VAR_INPUT
  ENCODER : DINT ;	//Positionswert Encoder
  INKR : DINT ;	//Inkremente für einen gezählten Wegimpuls (TEILUNG)
  FRG : BOOL ;	//Zählfreigabe
  RICHTUNG : BOOL ;	//Zählrichtung 0 = vorw. / 1 = rückw.
END_VAR
VAR_IN_OUT
  Weg : DINT ;	//Speicher für Wegwert
  tmpWeg : DINT ;	//Hilfsspeicher für Zwischenspeicherung Startwert Zählen
  tmpINKR : DINT ;
  btmpStart : BOOL ;	//Hilfsmerker Zähler gestartet
END_VAR
VAR_TEMP
  WEGDIFF : DINT ;
END_VAR
BEGIN
NETWORK
TITLE =

      UN    #FRG; // keine FRG
      R     #btmpStart; // Zähler gestartet clr
      BEB   ;

NETWORK
TITLE =Zähler starten: jedesmal bei Wiederkehr von FRG neu starten

      U     #btmpStart; // Zähler bereits gestartet
      SPB   NWE; // Netzwerkende

      S     #btmpStart; // Zähler ist gestartet

      L     #ENCODER; // Encoder-Wert
      T     #tmpWeg; // als Startwert speichern

      L     #INKR; // Anzahl der zu zählenden Inkremente
      T     #tmpINKR; // in temp-Varible speichern

NWE:  NOP   0;
NETWORK
TITLE =

      L     #ENCODER; // aktueller Encoder Wert
      L     #tmpWeg; // Hilfsspeicher StartWert Encoder
      -D    ; // zurückgelegte Strecke
      SPP   WEIT; // Wenn positiv dann weiter
      NEGD  ; // Vorzeichen drehen
WEIT: L     #tmpINKR; // Anzahl der Inkremente pro Wegeinheit
      -D    ; // >=0 : Wegeinheit erreicht; >0 zuviel gez. INKR
      SPPZ  CNT; // springe zu zählen, wenn >=0
      BEA   ;

CNT:  L     #INKR; // Inkremente pro Wegeinheit
      TAK   ; // zu viel gezählte INKR in Akku 1 zurück
      -D    ; // Korrektur SollInkr.: beim nächsten mal weniger zählen
      T     #tmpINKR; // beim nächsten mal zu zählende Inkremente

      L     1;
      UN    #RICHTUNG; // keine Richtungsumkehr
      SPB   INC; // Weg erhöhen
      NEGD  ; // Vorzeichen drehen
INC:  L     #Weg;
      +D    ;
      T     #Weg;

      L     #ENCODER; // Encoder-Wert
      T     #tmpWeg; // als Startwert speichern

END_FUNCTION

FUNCTION "m7b_AchseReferenzieren" : VOID
TITLE =Standard Funktion Achse referenzieren
//AUTOR: Stefan Maag, Dipl.-Ing. (FH) Elektrotechnik
//DATUM: 6/2003
//INTERNET: www.maagic7.de
//
//AENDERUNGSVERMERKE:
//--------------------------------------------------------------------------------
//DATUM        NAME       AENDERUNG
//--------------------------------------------------------------------------------
//07.04.2009   S.Maag     IO auf Ausgänge, REF_OK bei INIT/Reset löschen
//--------------------------------------------------------------------------------
//
//HINWEISE:
AUTHOR : 'S.Maag'
FAMILY : Maagic7
VERSION : 0.1


VAR_INPUT
  REF_START : BOOL ;	//Start rererenzieren
  REF_SENSOR : BOOL ;	//Referenzsensor 1-Position
  MSG_REF_VERLASSEN : BOOL ;	//Meldung Referenzpunkt ist verlassen
  RESET : BOOL ;
END_VAR
VAR_OUTPUT
  REF_OK : BOOL ;	//Achse ist Referenziert
  REF_FAHRT : BOOL ;	//Referenzfahrt aktiv! mit diesem Ausgang die Achse fahren
  REF_VERLASSEN : BOOL ;	//Steuerausgang Referenzpunkt verlassen
  ERROR : BOOL ;	//Fehler
END_VAR
VAR_IN_OUT
  IO_LOAD_POS : BOOL ;	//Referenzposition laden
  SNR : INT ;	//Schrittnummer
  tmpTime : TIME ;
END_VAR
VAR_TEMP
  SysTime : TIME ;
END_VAR
BEGIN
NETWORK
TITLE =Fehlerüberwachung, Zeitüberschreitung referenzieren

      L     #SNR; // Wenn Schrittnummer >1, dann ist
      L     1; // der Ablauf gestartet und Fehlerprüfung
      >I    ; // findet statt
      SPBN  NOER; // sonst kein Fehler

      CALL "TIME_TCK" (// aktuelle Systemzeit
           RET_VAL                  := #SysTime);// Zwischenspeichern

      L     #tmpTime; // gespeicherte Zeit: RefSensor erreicht
      L     #SysTime;
      UC    "m7b_ABS_DIFF_S7SysTime"; // Absolute Differenz S7SytemTimer 31Bit
      L     T#1M; // 30 sec
      >=D   ; // wenn 30 sec erreicht, dann Fehler
      SPB   ERR;

NOER: CLR   ; // kein Fehler
ERR:  =     #ERROR;
NETWORK
TITLE =RESET

      U     #RESET; // Schrittabläufe  clr
      SPBNB _001;
      L     0;
      T     #SNR;
_001: NOP   0;
NETWORK
TITLE =Ablauf Referenzieren: Ablaufsteuerung

      L     #SNR; // Schrittnummer
      SPL   CLR; // Sprungziel bei SNR>max
      SPA   INIT; // 0-Schritt, RESET
      SPA   S1; // Startschritt
      SPA   S2; // Schritt 2
      SPA   S3;
      SPA   S4;
      SPA   S5;

CLR:  L     1; // CLR : Ablauf löschen, RESET
      T     #SNR; // Schrittnummer auf Startschritt

      SET   ; // VKE = 1
// hier die bei RESET zu löschenden Merker eintragen
      R     #IO_LOAD_POS; // Referenzposition laden clr
      R     #REF_FAHRT; // Start Referenzfahrt
      R     #REF_VERLASSEN; // zuerst Referenzpunkt verlassen

      SPA   END;

INIT: SET   ; // Initialisierung, Null-Schritt
      R     #REF_OK;
      SPA   CLR;

NEXT: L     #SNR; // NEXT : Schrittnummer auf nächsten
      +     1; // Schritt
      T     #SNR;
END:  BEA   ;
NETWORK
TITLE =Warten auf Eingangssignal Referenzieren Start

S1:   U     #REF_START; // Eingangssignal referenzieren Start
      SPBN  END;

      R     #REF_OK; // Refernziert clr
      R     #IO_LOAD_POS; // Referenzposition laden clr
//   S     #OUT_REF_FAHRT              // Start Referenzfahrt
      S     #REF_VERLASSEN; // zuerst Referenzpunkt verlassen
      CALL "TIME_TCK" (// Systemzeit bei Ablauf start erreicht
           RET_VAL                  := #tmpTime);

      SPA   NEXT;

NETWORK
TITLE =Referenzpukt verlassen

S2:   U     #MSG_REF_VERLASSEN; // Meldung von aussen, Ref.Pkt. verlassen
      R     #REF_VERLASSEN; // zuerst Referenzpunkt verlassen
      S     #REF_FAHRT; // Start Referenzfahrt
      SPB   NEXT;
      SPA   END;
NETWORK
TITLE =Warten bis Referenzsensor erreicht

S3:   U     #REF_SENSOR; // Referenzsensor erreicht
      R     #REF_FAHRT; // Referenzfahrt clr
      SPBN  END;

      CALL "TIME_TCK" (// Systemzeit bei Referenzsensor erreicht
           RET_VAL                  := #tmpTime);

      SPA   NEXT;

NETWORK
TITLE =1 Sekunde Warten bis Achse steht, dann RefPos-laden

S4:   NOP   0;

      L     #tmpTime; // gespeicherte Zeit: RefSensor erreicht
      L     #SysTime; // aktuelle Systemzeit
      -D    ;
      SPP   PLUS;
      NEGD  ;
PLUS: L     T#1S; // 1 Sekunde
      >=D   ;
      SPBN  END;

      S     #IO_LOAD_POS; // Referenzposition laden

      SPA   NEXT;

NETWORK
TITLE =Referenzieren beendet, Referenzposition ist geladen

S5:   UN    #IO_LOAD_POS; // Merker Load_Pos ist 0, somit ist Position geladen
      S     #REF_OK;
      SPB   NEXT;
      SPA   END;

END_FUNCTION

FUNCTION "m7b_RPM_DRIVE" : VOID
TITLE =RPM Drive: Drehzahlberechnung Antrieb
//AUTOR: Stefan Maag, Dipl.-Ing. (FH) Elektrotechnik
//DATUM: 11/2017
//INTERNET: www.maagic7.de
//
//AENDERUNGSVERMERKE:
//--------------------------------------------------------------------------------
//DATUM        NAME        AENDERUNG
//--------------------------------------------------------------------------------
//16.08.2018   S.Maag     (Fmin => %Drehzahl) Berechnung hinzugefügt
//--------------------------------------------------------------------------------
//
//HINWEISE:
AUTHOR : 'S.Maag'
FAMILY : Maagic7
VERSION : 1.0


VAR_INPUT
  Sollwert : INT ;	//aktueller Sollwert Freuquenzumrichter % [0..1000]
  F_maxSoll : INT ;	//Frequenz [1/10Hz) bei Sollwert = 1000
  Fmin : INT ;	//untere Frequenzgrenze Motor (z.B. 30Hz ohne Fremdlüfter)
  MOT_Fnenn : INT ;	//Motor Nennfrequenz [Hz]
  MOT_Nnenn : INT ;	//Motor Nenndrehzahl [1/min]
  Igetr : REAL ;	//Übersetzung Getriebe
  Imasch : REAL ;	//Übersetung Maschine
END_VAR
VAR_OUTPUT
  F_Motor : INT ;	//Frequenz Motor
  N_MOT : INT ;	//Drehzahl Motor
  N_Masch : INT ;	//Drehzahl Maschine
  Prozent_Fmin : INT ;	//Drehzahl %, der Fmin entspricht
END_VAR
VAR_TEMP
  rSoll : REAL ;
  rF_MOT : REAL ;
  rN_MOT : REAL ;
END_VAR
BEGIN
NETWORK
TITLE =

      L     #Sollwert;
      ITD   ;
      DTR   ;
      T     #rSoll;
NETWORK
TITLE =Motorfrequenz

      L     #rSoll;
      L     1.000000e+003;
      /R    ;
      L     #F_maxSoll;
      ITD   ;
      DTR   ;
      *R    ;
      T     #rF_MOT;
      RND   ;
      T     #F_Motor;

NETWORK
TITLE =Motordrehzahl

      L     #rF_MOT;
      L     #MOT_Fnenn;
      ITD   ;
      DTR   ;
      /R    ;
      L     #MOT_Nnenn;
      ITD   ;
      DTR   ;
      *R    ;
      T     #rN_MOT;
      RND   ;
      T     #N_MOT;
NETWORK
TITLE =Maschinendrehzahl

      L     #Igetr;
      L     #Imasch;
      *R    ;
      L     #rN_MOT;
      *R    ;
      RND   ;
      T     #N_Masch;
NETWORK
TITLE =Fmin => %Drehzahl
//16.08.2018 S.Maag
//Fmin => Drehzahl hinzugefügt
      L     #Fmin;
      ITD   ;
      L     L#1000; // 1000%
      *D    ;
      L     #F_maxSoll;
      ITD   ;
      /D    ;
      T     #Prozent_Fmin;
END_FUNCTION

FUNCTION "m7b_MAPx4xBIT" : VOID
TITLE =4x mapping for BITs
//This function maps 4 individual Inputs to 4 individual Outputs using the
//mapping table MAP_1..MAP_4. There is no check for double using an INPUT.
//
//OUT(1)=IN(MAP_1)
//OUT(2)=IN(MAP_2)
//OUT(3)=IN(MAP_3)
//OUT(4)=IN(MAP_4)
//
//AUTOR: Stefan Maag, Dipl.-Ing. (FH) Elektrotechnik
//DATUM: 07/2012
//
//AENDERUNGSVERMERKE:
//--------------------------------------------------------------------------------
//DATUM        NAME       AENDERUNG
//--------------------------------------------------------------------------------
//25.06.2019   S.Maag     Bei MAP3 (NW4 Sprungmarke c4:) fehlte der CLR Befehl
//                        noch, so dass BIT 4 nicht immer korrekt durchgeschaltet
//                        wurde. Siehe Änderung vom 18.10.2012.
//                        Dieses Problem betrifft nur CPUs mit Interpreter.
//                        CPU's mit ASIC (VIPA, Siemens 318,400er)sind davon
//                        nicht betroffen!
//
//18.10.2012   S.Maag     Siemens CPU314C verarbeitet VKE bei Sprung nicht richtig
//                        wenn Sprungziel-Nr >1. Deswegen vor jedem U-Befehl ein
//                        CLR, somit werden alle Statusbits gelöscht und die
//                        Verknüpfung funktioniert bei allen Sprunziel-Nummern.
//--------------------------------------------------------------------------------
//HINWEISE:
//Seit 07.04.2020 neue Version in SCL mit 2 mapping modes.
//Für neue Projekte nur noch neue Version verwenden
AUTHOR : 'S.Maag'
FAMILY : Maagic7
VERSION : 0.1


VAR_INPUT
  IN_BIT_1 : BOOL ;
  IN_BIT_2 : BOOL ;
  IN_BIT_3 : BOOL ;
  IN_BIT_4 : BOOL ;
  MAP_1 : INT ;
  MAP_2 : INT ;
  MAP_3 : INT ;
  MAP_4 : INT ;
END_VAR
VAR_OUTPUT
  OUT_BIT_1 : BOOL ;
  OUT_BIT_2 : BOOL ;
  OUT_BIT_3 : BOOL ;
  OUT_BIT_4 : BOOL ;
END_VAR
VAR_TEMP
  iDIV : INT ;
END_VAR
BEGIN
NETWORK
TITLE =

      SET   ;
      SAVE  ;
      CLR   ;

NETWORK
TITLE =MAP 1 : OUT_BIT_1 := IN_BIT(MAP_1)
//18.10.2012   S.Maag
//bei Siemens CPU314C wird Zuweisung von Bit teilweise nicht korrekt verarbeitet,
//wenn in MAP ein Wert größer 1 steht. Bei 1 funktioniert es perfekt. Bei 2/3/4
//nicht.
      L     #MAP_1; // MAPPING-ZIEL Eingang 1
      SPL   a0; // Sprungziel bei MAP > 4
      SPA   a0; // MAP TO 0
      SPA   a1; // MAP TO 1
      SPA   a2; // MAP TO 2
      SPA   a3; // MAP TO 3
      SPA   a4; // MAO TO 4

a0:   CLR   ;
      SPA   aSAV;
a1:   CLR   ;
      U     #IN_BIT_1;
      SPA   aSAV;
a2:   CLR   ;
      U     #IN_BIT_2;
      SPA   aSAV;
a3:   CLR   ;
      U     #IN_BIT_3;
      SPA   aSAV;
a4:   CLR   ;
      U     #IN_BIT_4;
aSAV: =     #OUT_BIT_1;

NETWORK
TITLE =MAP 2 : OUT_BIT_2 := IN_BIT(MAP_2)

      L     #MAP_2; // MAPPING-ZIEL Eingang 2
      SPL   b0; // Sprungziel bei MAP > 4
      SPA   b0; // MAP TO 0
      SPA   b1; // MAP TO 1
      SPA   b2; // MAP TO 2
      SPA   b3; // MAP TO 3
      SPA   b4; // MAO TO 4

b0:   CLR   ;
      SPA   bSAV;
b1:   CLR   ;
      U     #IN_BIT_1;
      SPA   bSAV;
b2:   CLR   ;
      U     #IN_BIT_2;
      SPA   bSAV;
b3:   CLR   ;
      U     #IN_BIT_3;
      SPA   bSAV;
b4:   CLR   ;
      U     #IN_BIT_4;
bSAV: =     #OUT_BIT_2;

NETWORK
TITLE =MAP 3: OUT_BIT_3 := IN_BIT(MAP_3)

      L     #MAP_3; // MAPPING-ZIEL Eingang 3
      SPL   c0; // Sprungziel bei MAP > 4
      SPA   c0; // MAP TO 0
      SPA   c1; // MAP TO 1
      SPA   c2; // MAP TO 2
      SPA   c3; // MAP TO 3
      SPA   c4; // MAO TO 4

c0:   CLR   ;
      SPA   cSAV;
c1:   CLR   ;
      U     #IN_BIT_1;
      SPA   cSAV;
c2:   CLR   ;
      U     #IN_BIT_2;
      SPA   cSAV;
c3:   CLR   ;
      U     #IN_BIT_3;
      SPA   cSAV;
c4:   CLR   ;
      U     #IN_BIT_4;
cSAV: =     #OUT_BIT_3;

NETWORK
TITLE =MAP 4 : OUT_BIT_4 := IN_BIT(MAP_4)

      L     #MAP_4; // MAPPING-ZIEL Eingang 4
      SPL   d0; // Sprungziel bei MAP > 4
      SPA   d0; // MAP TO 0
      SPA   d1; // MAP TO 1
      SPA   d2; // MAP TO 2
      SPA   d3; // MAP TO 3
      SPA   d4; // MAO TO 4

d0:   CLR   ;
      SPA   dSAV;
d1:   CLR   ;
      U     #IN_BIT_1;
      SPA   dSAV;
d2:   CLR   ;
      U     #IN_BIT_2;
      SPA   dSAV;
d3:   CLR   ;
      U     #IN_BIT_3;
      SPA   dSAV;
d4:   CLR   ;
      U     #IN_BIT_4;
dSAV: =     #OUT_BIT_4;

NETWORK
TITLE =



END_FUNCTION

FUNCTION "m7b_X_Switch_BYTE" : VOID
TITLE =X_Switch_BYTE : Kreuzschalter für BYTE-Werte
//KREUZSCHALTUNG
//
//X_Switch : False: 1:1 - Schaltung OUT1:IN1; OUT2=IN2
//           True :   X - Schaltung OUT1:IN2; OUT2=IN1
//
//IN1 : Eingang 1
//IN2 : Eingang 2
//OUT1: Ausgang 1
//OUT2: Ausgang 2
//
//FC-ENO : Der X_Switch Eingang wird auf ENO druchgeschleift
//
//AUTOR: Stefan Maag, Dipl.-Ing. (FH) Elektrotechnik
//DATUM: 10/2013
//
//AENDERUNGSVERMERKE:
//--------------------------------------------------------------------------------
//DATUM        NAME            AENDERUNG
//--------------------------------------------------------------------------------
//
//--------------------------------------------------------------------------------
//
//HINWEISE: Entstand aus FC116 X_Switch_INT
AUTHOR : 'S.Maag'
FAMILY : Maagic7
VERSION : 0.1


VAR_INPUT
  X_Switch : BOOL ;	//False: 1:1 Schaltung; True: X-Schaltung
  IN1 : BYTE ;	//Eingangswert 1
  IN2 : BYTE ;	//Eingangswert 2
END_VAR
VAR_OUTPUT
  OUT1 : BYTE ;
  OUT2 : BYTE ;
END_VAR
BEGIN
NETWORK
TITLE =Kreuschalterfunktion

      U     #X_Switch; // Wenn Kreuzschaltung aktiv
      SAVE  ; // Schalter auf ENO durchschleifen
      SPB   X; // Ausgänge kreuz geschaltet

      L     #IN1; // Ausgänge 1:1 schalten
      T     #OUT1;

      L     #IN2;
      T     #OUT2;
      BEA   ;

X:    L     #IN1; // Ausgänge über Kreuz schalten
      T     #OUT2;

      L     #IN2;
      T     #OUT1;



END_FUNCTION

FUNCTION "m7b_GetBitFromByte" : VOID
TITLE =Bit mit Nr. aus Byte lesen; GetBit(IN_Byte, IN_BitNo)
//AUTOR: Stefan Maag, Dipl.-Ing. (FH) Elektrotechnik
//DATUM: 11/2015
//
//AENDERUNGSVERMERKE:
//--------------------------------------------------------------------------------
//DATUM        NAME         AENDERUNG
//--------------------------------------------------------------------------------
//22.04.2020   S.Maag       Code optimiert: Abfrage <0 & >0 durch AND 7
//                          ersetzt. Indirekte Adressierung durch SRW
//--------------------------------------------------------------------------------
VERSION : 0.1


VAR_INPUT
  IN_BYTE : BYTE ;
  IN_BitNo : INT ;	//Bit [0..7]
END_VAR
BEGIN
NETWORK
TITLE =%Byte.BitNo

      L     #IN_BitNo; // Bit-No
      UW    W#16#7; // Limit [0..7]
      +     1; // Add 1 because we must Shift 1 for Bit 0
      L     #IN_BYTE; // load the Byte
      SRW   ; // Shift right to get the selected bit
      U     >0; // IF BIT
      SAVE  ;
END_FUNCTION

FUNCTION "m7b_SetBitInByte" : BYTE
TITLE =Bit mit Nr. in Byte zuweisen; SetBit(BitVal,myByte, BitNo)
//
//ENO : Returns the original value of the selected Bit
//
//AUTOR: Stefan Maag, Dipl.-Ing. (FH) Elektrotechnik
//DATUM: 4/2020
//
//AENDERUNGSVERMERKE:
//--------------------------------------------------------------------------------
//DATUM        NAME         AENDERUNG
//--------------------------------------------------------------------------------
//
//--------------------------------------------------------------------------------
VERSION : 0.1


VAR_INPUT
  IN_BitVal : BOOL ;	//Bit value to set (FALSE, TRUE)
  IN_BYTE : BYTE ;
  IN_BitNo : INT ;	//Bit [0..7]
END_VAR
VAR_TEMP
  tmpByte : BYTE ;
  tmpBitNo : INT ;
END_VAR
BEGIN
NETWORK
TITLE =%Byte.BitNo := BitVal
//ENO := %In_BYTE.BitNo;
//
//tmpByte := IN_BYTE;
//%tmpByte.BitNo := IN_BitVal;
//RET_VAL := tmpByte;
      L     #IN_BitNo; // Bit-No
      UW    W#16#7; // Limit [0..7]
      T     #tmpBitNo; // BitNo 0..7

      L     #IN_BYTE; // Load IN_BYTE
      T     #tmpByte; // copy it to tmpByte

      L     P##tmpByte; // Pointer *Byte
      L     #tmpBitNo; // + BitNo
      +D    ; // = Pointer *Byte.BitNo
      LAR1  ; // Load *Byte.BitNo in AddressRegister 1

      U      [AR1,P#0.0]; // Get the original BitValue %IN_BYTE.BitNo
      SAVE  ; // ENO := %IN_BYTE.BitNo
      CLR   ;

      U     #IN_BitVal; // The BitValue (True or False)
      =      [AR1,P#0.0]; // *Byte.BitNo := BitVal
      L     #tmpByte; // The modified Byte
      T     #RET_VAL; // Return the modified Byte

END_FUNCTION

FUNCTION "m7b_RP_COPY_CHRONO" : VOID
TITLE =RP_COPY_CHRONO: kopiert Ringpuffer in choronologischer Folge
//Kopiert einen Ringpuffer. Die Daten werden dabei chronologisch in aufsteigender
//Reihenfolge angeordnet. D.h. am Anfang des Zieldatenbereichs steht der älteste
//Wert, am Ende der Neueste.
//
//AUTOR: Stefan Maag, Dipl.-Ing. (FH) Elektrotechnik
//DATUM: 1/2005
//INTERNET: www.maagic7.de
//
//AENDERUNGSVERMERKE:
//--------------------------------------------------------------------------------
//DATUM        NAME        AENDERUNG
//--------------------------------------------------------------------------------
//
//--------------------------------------------------------------------------------
//
//HINWEISE: getestet 10.01.2005
AUTHOR : 'S.Maag'
FAMILY : Maagic7
VERSION : 0.1


VAR_INPUT
  QUELL_DB : INT ;
  ZIEL_DB : INT ;
  QUELL_DW : INT ;
  ZIEL_DW : INT ;
  ANZAHL : INT ;
  ptrRP : INT ;
  RP_VOLL : BOOL ;
END_VAR
VAR_TEMP
  Quell_DB_Nr : INT ;
  Ziel_Db_Nr : INT ;
  QUELL_ADR : DINT ;
  ZIEL_ADR : DINT ;
  LOOP : INT ;
  ACTIVE_DI : INT ;	//Zwichenspeicher Nr. aktiver Instanzdatenbaustein
  AR1 : DWORD ;
  AR2 : DWORD ;
  END_ADR : DINT ;
  Quell_ADR_1 : DINT ;	//Quelladresse des 1. zu kopierenden Datenblocks
  Ziel_ADR_2 : DINT ;	//Zieladresse des 2. zu kopierenden Datenblocks
  ANZAHL1 : INT ;	//Anzahl DW des 1. zu kopierenden Blocks
  ANZAHL2 : INT ;	//Anzahl DW des 2. zu kopierenden Blocks
END_VAR
BEGIN
NETWORK
TITLE =Register sichern

      L     DINO; // Nr. Instanzdatenbaustein in AKKU
      T     #ACTIVE_DI;
      TAR1  #AR1; // Adressregister 1 sichern
      TAR2  #AR2; // Adressregister 2 sichern

NETWORK
TITLE =Datenbausteinnummern müssen auf Temp-Variablen kopiert werden

      L     #QUELL_DB;
      T     #Quell_DB_Nr;

      L     #ZIEL_DB;
      T     #Ziel_Db_Nr;
NETWORK
TITLE =Variablen initalisieren, bei welchen dies nötig ist

      L     0;
      T     #ANZAHL1;
      T     #ANZAHL2;

NETWORK
TITLE =Endadresse Quell-Datenbereich berechnen

      L     #QUELL_DW;
      L     #ANZAHL;
      SLW   1;
      +D    ;
      +     L#-2;
      T     #END_ADR;
NETWORK
TITLE =1. zu kopierender Datenblock
//Der 1. zu kopierende Datenblock enthält die älteseten Ringpufferdaten. Also
//alle Daten ab der Adresse des aktuellen Pointers (Pointer zeigt immer auf die
//Adresse des als nächstes zu schreibenden Wertes, die ist gleichzeitig der
//älteste Wert im Puffer)
//Ringpuffers.
      L     #ptrRP; // Pointer Ringpuffer (ByteAdresse)
      T     #Quell_ADR_1; // Stardadresse 1. zu kopierender Block

      L     #END_ADR; // Wenn END_ADR <= Pointer,
      L     #ptrRP; // dann kann kein hinterer
      -D    ;
      SRD   1; // halbieren, da Byteadressen
      T     #ANZAHL1; // Anzahl zu kopierender DW

NETWORK
TITLE =Adressen für Quell und Ziel-DW als Pointer in Adressregister

      L     #Quell_ADR_1; // Quelldatenwort-Nr
      SLD   3; // als Pointer
      L     P#0.0;
      +D    ;
      LAR1  ; // ins Adressregister 1

      L     #ZIEL_DW; // Zieldatenwort-Nr
      SLD   3; // als Pointer
      L     P#0.0;
      +D    ;
      LAR2  ; // ins Adressregister 2
NETWORK
TITLE =Daten kopieren
//Schnelle Kopierroutine: kopiert Blöcke von Datenworten in 4 Byte Schritten
//Quell- und Ziel- DB müssen nur einmal geöffnet werden.
      AUF   DI [#Quell_DB_Nr]; // Quell-DB als Instanz-DB öffnen
      AUF   DB [#Ziel_Db_Nr]; // Ziel-DB als Global-DB öffnen

      L     #ANZAHL1; // Anzahl der zu kopierenden DW's (Anzahl der 16 Bit-Werte)
      SRW   1; // in Anzahl der 32-Bit-Werte umrechen
LOOP: L     DID [AR1,P#0.0]; // Quell-DW lesen
      T     DBD [AR2,P#0.0]; // Ziel-DW lesen
      +AR1  P#4.0; // Quell-Pointer in AR1 um 4 Bytes erhöhen
      +AR2  P#4.0; // Ziel-Pointer in AR2 um 4 Bytes erhöhen
      TAK   ; // Schleifenzählr wieder in Akku 1 zurück
      LOOP  LOOP; // Schleifenzähler bearbeiten

      L     #ANZAHL1; // nun noch prüfen ob noch ein 16-Bit-Wert kopiert werden muss
      SRW   1; // LSB von Anzahl wird in Ergebnisvorzeichenregister geschoben
      SPZ   END; // prüft somit, ob LSB von ANZAHL = 1 ist
      L     DIW [AR1,P#0.0]; // Dann muss das letze DW noch kopiert werden
      T     DBW [AR2,P#0.0];
NETWORK
TITLE =Anzahl Datenworte des 2. zu kopierenden Blocks

      NOP   0;
      L     #ANZAHL; // gesamte Anzahl zu kopierender Datenworte
      L     #ANZAHL1; // Anzahl der im 1. Durchgang kopierten Datenworte
      -I    ; //
      T     #ANZAHL2; // Anzahl der im 2. Durchgang zu kopierenden Worte
      SPMZ  END; // springt zum Ende, wenn Ergebnis <=0

NETWORK
TITLE =Zieladresse 2. zu kopierender Block

      L     #ANZAHL1; // Anzahl Datenworte
      L     #ZIEL_DW;
      +I    ; // Anzahl 2x zu Ziel_DW zählen
      +I    ; // wegen Byteadressen
      T     #Ziel_ADR_2;
NETWORK
TITLE =Adressen für Quell und Ziel-DW als Pointer in Adressregister

      L     #QUELL_DW; // Quelldatenwort-Nr
      SLD   3; // als Pointer
      L     P#0.0;
      +D    ;
      LAR1  ; // ins Adressregister 1

      L     #Ziel_ADR_2; // Zieldatenwort-Nr
      SLD   3; // als Pointer
      L     P#0.0;
      +D    ;
      LAR2  ; // ins Adressregister 2
NETWORK
TITLE =Daten kopieren

      AUF   DI [#Quell_DB_Nr]; // Quell-DB als Instanz-DB öffnen
      AUF   DB [#Ziel_Db_Nr]; // Ziel-DB als Global-DB öffnen

      L     #ANZAHL2; // Anzahl der zu kopierenden DW's (Anzahl der 16 Bit-Werte)
      SRW   1; // in Anzahl der 32-Bit-Werte umrechen
LP2:  L     DID [AR1,P#0.0]; // Quell-DW lesen
      T     DBD [AR2,P#0.0]; // Ziel-DW lesen
      +AR1  P#4.0; // Quell-Pointer in AR1 um 4 Bytes erhöhen
      +AR2  P#4.0; // Ziel-Pointer in AR2 um 4 Bytes erhöhen
      TAK   ; // Schleifenzählr wieder in Akku 1 zurück
      LOOP  LP2; // Schleifenzähler bearbeiten

      L     #ANZAHL2; // nun noch prüfen ob noch ein 16-Bit-Wert kopiert werden muss
      SRW   1; // LSB von Anzahl wird in Ergebnisvorzeichenregister geschoben
      SPZ   END; // prüft somit, ob LSB von ANZAHL = 1 ist
      L     DIW [AR1,P#0.0]; // Dann muss das letze DW noch kopiert werden
      T     DBW [AR2,P#0.0];
NETWORK
TITLE =Registerinhalte wieder herstellen

END:  AUF   DI [#ACTIVE_DI]; // Activen Instanz-DB wieder herstellen
      LAR1  #AR1; // Adressregister 1 wieder herstellen
      LAR2  #AR2; // Adressregister 2 wieder herstellen

      SET   ;
      SAVE  ;
      CLR   ;
END_FUNCTION

FUNCTION "m7b_ChangeEvent_INT" : VOID
TITLE =Ereignis INT Wert hat sich geändert
//Der FC-ENO-Ausgang wird für einen Zyklus "1", wenn der sich der Eingangswert
//geändert hat, ansonsten ist der FC-ENO-Ausgang "0"
//
//AUTOR: Stefan Maag, Dipl.-Ing. (FH) Elektrotechnik
//DATUM: 8/2008
//INTERNET: www.maagic7.de
//
//AENDERUNGSVERMERKE:
//--------------------------------------------------------------------------------
//DATUM        NAME            AENDERUNG
//--------------------------------------------------------------------------------
//
//--------------------------------------------------------------------------------
//
//HINWEISE:
AUTHOR : 'S.Maag'
FAMILY : Maagic7
VERSION : 0.1


VAR_INPUT
  inINT : INT ;
END_VAR
VAR_IN_OUT
  memINT : INT ;
END_VAR
BEGIN
NETWORK
TITLE =

      L     #inINT; // Eingangwert
      L     #memINT; // letzter Wert
      <>I   ; // ungleich!
      SAVE  ; // als ENO ausgeben
      SPB   do; // und neuen
      BEA   ;
do:   L     #inINT; // Wert speichern
      T     #memINT;

END_FUNCTION

FUNCTION "m7b_RP_WRITE_INT" : VOID
TITLE =Ringpuffer schreiben INT-Werte
//AUTOR: Stefan Maag, Dipl.-Ing. (FH) Elektrotechnik
//DATUM: 7/2008
//INTERNET: www.maagic7.de
//
//AENDERUNGSVERMERKE:
//--------------------------------------------------------------------------------
//DATUM        NAME        AENDERUNG
//--------------------------------------------------------------------------------
//09.07.2010   S.Maag      ENO nur True, wenn Ringpuffer geschrieben/verarbeitet
//                         wird, sonst FALSE
//--------------------------------------------------------------------------------
//
//HINWEISE:
AUTHOR : 'S.Maag'
FAMILY : Maagic7
VERSION : 0.1


VAR_INPUT
  DB_RP : BLOCK_DB ;
  RP_POS : BOOL ;	//Ringpuffer schreiben positiv
  RP_NEG : BOOL ;	//Ringpuffer schreiben negativ
  IN_INT : INT ;	//Eingangswert INT
END_VAR
VAR_IN_OUT
  RP_IDX : INT ;	//Indexwert Ringpuffer 0..255
END_VAR
VAR_TEMP
  AR1 : DWORD ;
END_VAR
BEGIN
NETWORK
TITLE =

      TAR1  #AR1; // Adressregister 1 sichern

NETWORK
TITLE =

      U     #RP_POS; // positiver Impuls := Ringpuffer vorwärts
      SPB   pos;

      U     #RP_NEG; // negativer Impuls := Ringpuffer rückwärts
      SPB   neg;

      CLR   ; // ENO = FALSE, => keine Verarbeitung
      SAVE  ;
      BEA   ;

pos:  L     #RP_IDX; // positiver Impuls := Ringpuffer vorwärts
      INC   1; // INC: Bytebefehl 0..255
      SPA   save;

neg:  L     #RP_IDX; // negativer Impuls := Ringpuffer rückwärts
      DEC   1; // DEC: Bytebefehl 0..255

save: T     #RP_IDX; // Indexwert Ringpuffer 0..255
      SLD   4; // SLD 1 wegen DINT-Werten=>Byte + SLD 3 wegen Pointer
      L     P#0.0; // 0-Pointer addieren
      +D    ; // Pointer auf Daten erzeugen
      LAR1  ; // in Adressregister 1 laden

      AUF   #DB_RP; // Ringpuffer DB öffnen
      L     #IN_INT; // Eingangswert laden
      T     DBW [AR1,P#0.0]; // in DB speichern

      LAR1  #AR1; // ursprüngliches Adressregister 1 herstellen
      SET   ; // ENO = TRUE, => Verarbeitung
      SAVE  ;
      BEA   ;


END_FUNCTION

FUNCTION "m7b_RP_READ_INT" : INT
TITLE =Ringpuffer lesen INT-Werte
//AUTOR: Stefan Maag, Dipl.-Ing. (FH) Elektrotechnik
//DATUM: 7/2008
//INTERNET: www.maagic7.de
//
//AENDERUNGSVERMERKE:
//--------------------------------------------------------------------------------
//DATUM        NAME        AENDERUNG
//--------------------------------------------------------------------------------
//
//--------------------------------------------------------------------------------
//
//HINWEISE:
AUTHOR : 'S.Maag'
FAMILY : Maagic7
VERSION : 0.1


VAR_INPUT
  DB_RP : BLOCK_DB ;
  RP_IDX : INT ;	//Ringpuffer Index
  RP_OFFSET : INT ;	//Offeset Ringpufferindex
END_VAR
VAR_TEMP
  AR1 : DWORD ;
END_VAR
BEGIN
NETWORK
TITLE =

      TAR1  #AR1; // Adressregister 1 sichern

      L     #RP_IDX; // aktueller Ringpuffer-Index
      L     #RP_OFFSET; // Offset für lesen
      -I    ;
      L     W#16#FF; // auf 0..255 begrenzen
      UW    ;
      SLD   4; // SLD 1 wegen DINT-Werten=>Byte + SLD 3 wegen Pointer
      L     P#0.0; // 0-Pointer addieren
      +D    ; // Pointer auf Daten erzeugen
      LAR1  ; // in Adressregister 1 laden

      AUF   #DB_RP; // Ringpuffer DB öffnen
      L     DBW [AR1,P#0.0]; // Wert aus Ringpuffer laden
      T     #RET_VAL; // Rückgabewert

      LAR1  #AR1; // ursprüngliches Adressregister 1 herstellen
      SET   ;
      SAVE  ;
      CLR   ;

END_FUNCTION

FUNCTION "m7b_MUXx3xINT" : INT
TITLE =3-fach Integer Multiplexer
//AUTOR: Stefan Maag, Dipl.-Ing. (FH) Elektrotechnik
//DATUM: 8/2003
//INTERNET: www.maagic7.de
//
//AENDERUNGSVERMERKE:
//--------------------------------------------------------------------------------
//DATUM        NAME        AENDERUNG
//--------------------------------------------------------------------------------
//24.04.2009   S.Maag      EN0 := Signal Wert selektiert
//                               (S1 | S2 | S3)  AND ENABLE
//
//29.01.2013   S.Maag      Anzeige aktiver Kanal (DSP_CHANNEL)
//--------------------------------------------------------------------------------
//
//HINWEISE:
AUTHOR : 'S.Maag'
FAMILY : Maagic7
VERSION : 2.0


VAR_INPUT
  S1 : BOOL ;
  S2 : BOOL ;
  S3 : BOOL ;
  ENABLE : BOOL ;
  INT1 : INT ;
  INT2 : INT ;
  INT3 : INT ;
END_VAR
VAR_OUTPUT
  DSP_CHANNEL : INT ;	//Displays the activated channel
END_VAR
BEGIN
NETWORK
TITLE =

      UN    #ENABLE; // keine Freigabe, dann 0 ausgeben
      SPB   STOP;

      U     #S1;
      SPB   S1;
      U     #S2;
      SPB   S2;
      U     #S3;
      SPB   S3;

      SPA   STOP;

S1:   L     1; // Wert für Kanalanzeige
      L     #INT1;
      SPA   SAVE;

S2:   L     2;
      L     #INT2;
      SPA   SAVE;

S3:   L     3;
      L     #INT3;
      SPA   SAVE;

STOP: CLR   ; // EN0-Ausgang =0, da Stopp
      L     0; // Wert für Kanalanzeige
      L     0; // Wert für Multiplexer

SAVE: SAVE  ;
      T     #RET_VAL; // Mulitplexer Ausgang
      TAK   ; // Wert aktiver Kanal
      T     #DSP_CHANNEL; // Anzeige aktiver Kanal


END_FUNCTION

FUNCTION "m7b_MUXx4xINT" : INT
TITLE =4-fach Integer Multiplexer
//AUTOR: Stefan Maag, Dipl.-Ing. (FH) Elektrotechnik
//DATUM: 8/2008
//INTERNET: www.maagic7.de
//
//AENDERUNGSVERMERKE:
//--------------------------------------------------------------------------------
//DATUM        NAME        AENDERUNG
//--------------------------------------------------------------------------------
//25.08.2008   S.Maag      enstanden aus MUXx3xINT
//
//24.04.2009   S.Maag      EN0 := Signal Wert selektiert
//                               (S1 | S2 | S3)  AND ENABLE
//
//29.01.2013   S.Maag      Anzeige aktiver Kanal (DSP_CHANNEL)
//--------------------------------------------------------------------------------
//
//HINWEISE:
AUTHOR : 'S.Maag'
FAMILY : Maagic7
VERSION : 2.0


VAR_INPUT
  S1 : BOOL ;
  S2 : BOOL ;
  S3 : BOOL ;
  S4 : BOOL ;
  ENABLE : BOOL ;
  INT1 : INT ;
  INT2 : INT ;
  INT3 : INT ;
  INT4 : INT ;
END_VAR
VAR_OUTPUT
  DSP_CHANNEL : INT ;	//Displays the activated channel
END_VAR
BEGIN
NETWORK
TITLE =

      UN    #ENABLE; // keine Freigabe, dann 0 ausgeben
      SPB   STOP;

      U     #S1;
      SPB   S1;
      U     #S2;
      SPB   S2;
      U     #S3;
      SPB   S3;
      U     #S4;
      SPB   S4;

      SPA   STOP;

S1:   L     1; // Wert für Kanalanzeige
      L     #INT1;
      SPA   SAVE;

S2:   L     2;
      L     #INT2;
      SPA   SAVE;

S3:   L     3;
      L     #INT3;
      SPA   SAVE;

S4:   L     4;
      L     #INT4;
      SPA   SAVE;

STOP: CLR   ; // EN0-Ausgang =0, da Stopp
      L     0; // Wert für Kanalanzeige
      L     0; // Wert für Multiplexer

SAVE: SAVE  ;
      T     #RET_VAL; // Mulitplexer Ausgang
      TAK   ; // Wert aktiver Kanal
      T     #DSP_CHANNEL; // Anzeige aktiver Kanal

END_FUNCTION

FUNCTION "m7b_MAPx4xINT" : VOID
TITLE =4x mapping for INTEGER
//This function maps 4 individual Inputs to 4 individual Outputs using the
//mapping table MAP_1..MAP_4. There is no check for double using an INPUT.
//
//OUT(1)=IN(MAP_1)
//OUT(2)=IN(MAP_2)
//OUT(3)=IN(MAP_3)
//OUT(4)=IN(MAP_4)
//
//AUTOR: Stefan Maag, Dipl.-Ing. (FH) Elektrotechnik
//DATUM: 07/2012
//
//AENDERUNGSVERMERKE:
//--------------------------------------------------------------------------------
//DATUM        NAME       AENDERUNG
//--------------------------------------------------------------------------------
//
//--------------------------------------------------------------------------------
//HINWEISE:
//Seit 07.04.2020 neue Version in SCL mit 2 mapping Modes.
//Für neue Projekte nur noch neue Version verwenden
AUTHOR : 'S.Maag'
FAMILY : Maagic7
VERSION : 0.1


VAR_INPUT
  IN_1 : INT ;	//Input Value 1
  IN_2 : INT ;	//Input Value 2
  IN_3 : INT ;	//Input Value 3
  IN_4 : INT ;	//Input Value 4
  ZERO_VAL : INT ;	//Zero Value (used as 'zero', if no mapping)
  MAP_1 : INT ;	//Source Nr. for OUT_1: OUT_1=IN(MAP_1)
  MAP_2 : INT ;	//Source Nr. for OUT_2: OUT_2=IN(MAP_2)
  MAP_3 : INT ;	//Source Nr. for OUT_3: OUT_3=IN(MAP_3)
  MAP_4 : INT ;	//Source Nr. for OUT_4: OUT_3=IN(MAP_4)
END_VAR
VAR_OUTPUT
  OUT_1 : INT ;
  OUT_2 : INT ;
  OUT_3 : INT ;
  OUT_4 : INT ;
END_VAR
BEGIN
NETWORK
TITLE =

      SET   ;
      SAVE  ;
      CLR   ;

NETWORK
TITLE =MAP 1 : OUT_1 := IN (MAP_1)

      L     #MAP_1; // MAPPING-ZIEL Eingang 1
      SPL   a0; // Sprungziel bei MAP > 4
      SPA   a0; // MAP TO 0
      SPA   a1; // MAP TO 1
      SPA   a2; // MAP TO 2
      SPA   a3; // MAP TO 3
      SPA   a4; // MAO TO 4

a0:   L     #ZERO_VAL;
      SPA   aSAV;
a1:   L     #IN_1;
      SPA   aSAV;
a2:   L     #IN_2;
      SPA   aSAV;
a3:   L     #IN_3;
      SPA   aSAV;
a4:   L     #IN_4;
aSAV: T     #OUT_1;
NETWORK
TITLE =MAP 2 : OUT_2 := IN (MAP_2)

      L     #MAP_2; // MAPPING-ZIEL Eingang 2
      SPL   b0; // Sprungziel bei MAP > 4
      SPA   b0; // MAP TO 0
      SPA   b1; // MAP TO 1
      SPA   b2; // MAP TO 2
      SPA   b3; // MAP TO 3
      SPA   b4; // MAO TO 4

b0:   L     #ZERO_VAL;
      SPA   bSAV;
b1:   L     #IN_1;
      SPA   bSAV;
b2:   L     #IN_2;
      SPA   bSAV;
b3:   L     #IN_3;
      SPA   bSAV;
b4:   L     #IN_4;
bSAV: T     #OUT_2;
NETWORK
TITLE =MAP 3 : OUT_3 := IN (MAP_3)

      L     #MAP_3; // MAPPING-ZIEL Eingang 3
      SPL   c0; // Sprungziel bei MAP > 4
      SPA   c0; // MAP TO 0
      SPA   c1; // MAP TO 1
      SPA   c2; // MAP TO 2
      SPA   c3; // MAP TO 3
      SPA   c4; // MAO TO 4

c0:   L     #ZERO_VAL;
      SPA   cSAV;
c1:   L     #IN_1;
      SPA   cSAV;
c2:   L     #IN_2;
      SPA   cSAV;
c3:   L     #IN_3;
      SPA   cSAV;
c4:   L     #IN_4;
cSAV: T     #OUT_3;
NETWORK
TITLE =MAP 4 : OUT_4 := IN (MAP_4)

      L     #MAP_4; // MAPPING-ZIEL Eingang 4
      SPL   d0; // Sprungziel bei MAP > 4
      SPA   d0; // MAP TO 0
      SPA   d1; // MAP TO 1
      SPA   d2; // MAP TO 2
      SPA   d3; // MAP TO 3
      SPA   d4; // MAO TO 4

d0:   L     #ZERO_VAL;
      SPA   dSAV;
d1:   L     #IN_1;
      SPA   dSAV;
d2:   L     #IN_2;
      SPA   dSAV;
d3:   L     #IN_3;
      SPA   dSAV;
d4:   L     #IN_4;
dSAV: T     #OUT_4;
END_FUNCTION

FUNCTION "m7b_X_Switch_INT" : VOID
TITLE =X_Switch_INT : Kreuzschalter für INT-Werte
//KREUZSCHALTUNG
//
//X_Switch : False: 1:1 - Schaltung OUT1:IN1; OUT2=IN2
//           True :   X - Schaltung OUT1:IN2; OUT2=IN1
//
//IN1 : Eingang 1
//IN2 : Eingang 2
//OUT1: Ausgang 1
//OUT2: Ausgang 2
//
//FC-ENO : Der X_Switch Eingang wird auf ENO druchgeschleift
//
//AUTOR: Stefan Maag, Dipl.-Ing. (FH) Elektrotechnik
//DATUM: 03/2009
//INTERNET: www.maagic7.de
//
//AENDERUNGSVERMERKE:
//--------------------------------------------------------------------------------
//DATUM        NAME            AENDERUNG
//--------------------------------------------------------------------------------
//
//--------------------------------------------------------------------------------
//
//HINWEISE:
AUTHOR : 'S.Maag'
FAMILY : Maagic7
VERSION : 0.1


VAR_INPUT
  X_Switch : BOOL ;	//False: 1:1 Schaltung; True: X-Schaltung
  IN1 : INT ;	//Eingangswert 1
  IN2 : INT ;	//Eingangswert 2
END_VAR
VAR_OUTPUT
  OUT1 : INT ;
  OUT2 : INT ;
END_VAR
BEGIN
NETWORK
TITLE =Kreuschalterfunktion

      U     #X_Switch; // Wenn Kreuzschaltung aktiv
      SAVE  ; // Schalter auf ENO durchschleifen
      SPB   X; // Ausgänge kreuz geschaltet

      L     #IN1; // Ausgänge 1:1 schalten
      T     #OUT1;

      L     #IN2;
      T     #OUT2;
      BEA   ;

X:    L     #IN1; // Ausgänge über Kreuz schalten
      T     #OUT2;

      L     #IN2;
      T     #OUT1;



END_FUNCTION

FUNCTION "m7b_InvertRange_INT" : INT
TITLE =InvertRange_INT: Invertiert einen Bereich (Messrichtungsumkehr)
//Invertiert einen Wertebereich (Messrichtungsumkehr), vertauscht sozusagen Ober-
//und Untergrenze.
//Bei symetrischen Wertebereichen: MIN = -MAX ist das einfach eine
//Vorzeichenumkehr.
//
//ENO : Übersteuerungsanzeige: der invertierte Wert liegt ausserhalb des
//      Wertebereichs. Dieses Signal kann z.B. dazu verwendet werden um
//      eine gesonderte verarbeitung im Fehlerfalle druchzuführen.
//
//
//z.B. MIN=-100 MAX=100 VALUE=20 : Xinv= -20
//     MIN=  20 MAX=100 VALUE=20 : Xinv= 100
//                      VALUE=50 : Xinv=  70
//
//Xinv= MIN + MAX - VALUE
//
//
//AUTOR: Stefan Maag, Dipl.-Ing. (FH) Elektrotechnik
//DATUM: 10/2008
//INTERNET: www.maagic7.de
//
//AENDERUNGSVERMERKE:
//--------------------------------------------------------------------------------
//DATUM        NAME            AENDERUNG
//--------------------------------------------------------------------------------
//
//--------------------------------------------------------------------------------
//
//HINWEISE:
AUTHOR : 'S.Maag'
FAMILY : Maagic7
VERSION : 0.1


VAR_INPUT
  VALUE : INT ;	//Value to invert
  MIN : INT ;	//Minimum of Range
  MAX : INT ;	//Maximum of Range
END_VAR
BEGIN
NETWORK
TITLE =Invert Range: Wertebereich umkehren
//Xinv= MAX - VALUE + MIN  :  Bessere Berechnung wegen Überläufen
      L     #MAX;
      L     #VALUE;
      -I    ;
      L     #MIN;
      +I    ;
      T     #RET_VAL;
NETWORK
TITLE =FC-ENO-Ausgang als Übersteuerungsanzeige

      L     #MAX; // Maximalwert
      >I    ; // Wert > MAX
      SPB   SAVE; // Max-Wert überschritten
      TAK   ; // Ausgangswert in Akku 1 zurueck
      L     #MIN;
      <I    ;
      SPB   SAVE; // MinWert unterschritten
      CLR   ;
SAVE: SAVE  ;
      CLR   ;
END_FUNCTION

FUNCTION "m7b_MinDiffABS_INT" : VOID
TITLE =MinDiffABS_INT: Minimale Absolutdifferenz 2er INT-Werte ok!
//Überprüft, ob die absolute Differenz (absolut) zweier INT dem angebegenen
//Mindestwert entspricht. Wenn ja, dann wird ENO=True
//
//BENÖTIGTE SFCs: keine
//
//AUTOR: Stefan Maag, Dipl.-Ing. (FH) Elektrotechnik
//DATUM: 8/2008
//INTERNET: www.maagic7.de
//
//AENDERUNGSVERMERKE:
//--------------------------------------------------------------------------------
//DATUM        NAME        AENDERUNG
//--------------------------------------------------------------------------------
//10.09.2020   S.Maag      Ausgang iDiff hinzugefügt
//--------------------------------------------------------------------------------
//
//HINWEISE:
AUTHOR : 'S.Maag'
FAMILY : Maagic7
VERSION : 0.1


VAR_INPUT
  VAL_1 : INT ;
  VAL_2 : INT ;
  MinDiff : INT ;
END_VAR
VAR_OUTPUT
  iDiff : INT ;	//Differenz=ABS(VAL_1-VAL_2)
END_VAR
VAR_TEMP
  aktSysTime : TIME ;	//aktuelle Systemzeit
END_VAR
BEGIN
NETWORK
TITLE =prüfen ob Differenz ok

      L     #VAL_1;
      L     #VAL_2;
      -I    ;
      SPP   pos;
      NEGI  ;
pos:  T     #iDiff;
      L     #MinDiff;
      >=I   ;
      SAVE  ;

END_FUNCTION

FUNCTION "m7b_ChangeEvent_DINT" : VOID
TITLE =Ereignis DINT Wert hat sich geändert
//Der FC-ENO-Ausgang wird für einen Zyklus "1", wenn der sich der Eingangswert
//geändert hat, ansonsten ist der FC-ENO-Ausgang "0"
//
//AUTOR: Stefan Maag, Dipl.-Ing. (FH) Elektrotechnik
//DATUM: 8/2008
//INTERNET: www.maagic7.de
//
//AENDERUNGSVERMERKE:
//--------------------------------------------------------------------------------
//DATUM        NAME            AENDERUNG
//--------------------------------------------------------------------------------
//
//--------------------------------------------------------------------------------
//
//HINWEISE:
AUTHOR : 'S.Maag'
FAMILY : Maagic7
VERSION : 0.1


VAR_INPUT
  inDINT : DINT ;
END_VAR
VAR_IN_OUT
  memDINT : DINT ;
END_VAR
BEGIN
NETWORK
TITLE =

      L     #inDINT; // Eingangwert
      L     #memDINT; // letzter Wert
      <>D   ; // ungleich!
      SAVE  ; // als ENO ausgeben
      SPB   do; // und neuen
      BEA   ;
do:   L     #inDINT; // Wert speichern
      T     #memDINT;

END_FUNCTION

FUNCTION "m7b_RP_WRITE_DINT" : VOID
TITLE =Ringpuffer schreiben DINT-Werte
//AUTOR: Stefan Maag, Dipl.-Ing. (FH) Elektrotechnik
//DATUM: 7/2008
//INTERNET: www.maagic7.de
//
//AENDERUNGSVERMERKE:
//--------------------------------------------------------------------------------
//DATUM        NAME        AENDERUNG
//--------------------------------------------------------------------------------
//09.07.2010   S.Maag      ENO nur True, wenn Ringpuffer geschrieben/verarbeitet
//                         wird, sonst FALSE
//--------------------------------------------------------------------------------
//
//HINWEISE:
AUTHOR : 'S.Maag'
FAMILY : Maagic7
VERSION : 0.1


VAR_INPUT
  DB_RP : BLOCK_DB ;
  RP_POS : BOOL ;	//Ringpuffer schreiben positiv
  RP_NEG : BOOL ;	//Ringpuffer schreiben negativ
  IN_DINT : DINT ;	//Eingangswert DINT
END_VAR
VAR_IN_OUT
  RP_IDX : INT ;	//Indexwert Ringpuffer 0..255
END_VAR
VAR_TEMP
  AR1 : DWORD ;
END_VAR
BEGIN
NETWORK
TITLE =

      TAR1  #AR1; // Adressregister 1 sichern

NETWORK
TITLE =

      U     #RP_POS; // positiver Impuls := Ringpuffer vorwärts
      SPB   pos;

      U     #RP_NEG; // negativer Impuls := Ringpuffer rückwärts
      SPB   neg;

      CLR   ; // ENO = FALSE, => keine Verarbeitung
      SAVE  ;
      BEA   ;

pos:  L     #RP_IDX; // positiver Impuls := Ringpuffer vorwärts
      INC   1; // INC: Bytebefehl 0..255
      SPA   save;

neg:  L     #RP_IDX; // negativer Impuls := Ringpuffer rückwärts
      DEC   1; // DEC: Bytebefehl 0..255

save: T     #RP_IDX; // Indexwert Ringpuffer 0..255
      SLD   5; // SLD 2 wegen DINT-Werten=>Byte + SLD 3 wegen Pointer
      L     P#0.0; // 0-Pointer addieren
      +D    ; // Pointer auf Daten erzeugen
      LAR1  ; // in Adressregister 1 laden

      AUF   #DB_RP; // Ringpuffer DB öffnen
      L     #IN_DINT; // Eingangswert laden
      T     DBD [AR1,P#0.0]; // in DB speichern

      LAR1  #AR1; // ursprüngliches Adressregister 1 herstellen
      SET   ; // ENO = TRUE, => Verarbeitung
      SAVE  ;
      BEA   ;


END_FUNCTION

FUNCTION "m7b_RP_READ_DINT" : DINT
TITLE =Ringpuffer lesen DINT-Werte
//AUTOR: Stefan Maag, Dipl.-Ing. (FH) Elektrotechnik
//DATUM: 7/2008
//INTERNET: www.maagic7.de
//
//AENDERUNGSVERMERKE:
//--------------------------------------------------------------------------------
//DATUM        NAME        AENDERUNG
//--------------------------------------------------------------------------------
//
//--------------------------------------------------------------------------------
//
//HINWEISE:
AUTHOR : 'S.Maag'
FAMILY : Maagic7
VERSION : 0.1


VAR_INPUT
  DB_RP : BLOCK_DB ;
  RP_IDX : INT ;	//Ringpuffer Index
  RP_OFFSET : INT ;	//Offeset Ringpufferindex
END_VAR
VAR_TEMP
  AR1 : DWORD ;
END_VAR
BEGIN
NETWORK
TITLE =

      TAR1  #AR1; // Adressregister 1 sichern

      L     #RP_IDX; // aktueller Ringpuffer-Index
      L     #RP_OFFSET; // Offset für lesen
      -I    ;
      L     W#16#FF; // auf 0..255 begrenzen
      UW    ;
      SLD   5; // SLD 2 wegen DINT-Werten=>Byte + SLD 3 wegen Pointer
      L     P#0.0; // 0-Pointer addieren
      +D    ; // Pointer auf Daten erzeugen
      LAR1  ; // in Adressregister 1 laden

      AUF   #DB_RP; // Ringpuffer DB öffnen
      L     DBD [AR1,P#0.0]; // Wert aus Ringpuffer laden
      T     #RET_VAL; // Rückgabewert

      LAR1  #AR1; // ursprüngliches Adressregister 1 herstellen
      SET   ;
      SAVE  ;
      CLR   ;

END_FUNCTION

FUNCTION "m7b_MUXx3xDINT" : DINT
TITLE =3-fach DINT Multiplexer
//AUTOR: Stefan Maag, Dipl.-Ing. (FH) Elektrotechnik
//DATUM: 8/2003
//INTERNET: www.maagic7.de
//
//AENDERUNGSVERMERKE:
//--------------------------------------------------------------------------------
//DATUM        NAME        AENDERUNG
//--------------------------------------------------------------------------------
//24.04.2009   S.Maag      EN0 := Signal Wert selektiert
//                               (S1 | S2 | S3)  AND ENABLE
//
//29.01.2013   S.Maag      Anzeige aktiver Kanal (DSP_CHANNEL)
//--------------------------------------------------------------------------------
//
//HINWEISE:
AUTHOR : 'S.Maag'
FAMILY : Maagic7
VERSION : 2.0


VAR_INPUT
  S1 : BOOL ;
  S2 : BOOL ;
  S3 : BOOL ;
  ENABLE : BOOL ;
  DINT1 : DINT ;
  DINT2 : DINT ;
  DINT3 : DINT ;
END_VAR
VAR_OUTPUT
  DSP_CHANNEL : INT ;	//Displays the activated channel
END_VAR
BEGIN
NETWORK
TITLE =

      UN    #ENABLE; // keine Freigabe, dann 0 ausgeben
      SPB   STOP;

      U     #S1;
      SPB   S1;
      U     #S2;
      SPB   S2;
      U     #S3;
      SPB   S3;

      SPA   STOP;

S1:   L     1; // Wert für Kanalanzeige
      L     #DINT1;
      SPA   SAVE;

S2:   L     2;
      L     #DINT2;
      SPA   SAVE;

S3:   L     3;
      L     #DINT3;
      SPA   SAVE;

STOP: CLR   ; // EN0-Ausgang =0, da Stopp
      L     0; // Wert für Kanalanzeige
      L     L#0; // Wert für Multiplexer

SAVE: SAVE  ;
      T     #RET_VAL; // Mulitplexer Ausgang
      TAK   ; // Wert aktiver Kanal
      T     #DSP_CHANNEL; // Anzeige aktiver Kanal

END_FUNCTION

FUNCTION "m7b_MUXx4xDINT" : DINT
TITLE =4-fach DINT Multiplexer
//AUTOR: Stefan Maag, Dipl.-Ing. (FH) Elektrotechnik
//DATUM: 8/2008
//INTERNET: www.maagic7.de
//
//AENDERUNGSVERMERKE:
//--------------------------------------------------------------------------------
//DATUM        NAME        AENDERUNG
//--------------------------------------------------------------------------------
//25.08.2008   S.Maag      enstanden aus MUXx3xINT
//
//24.04.2009   S.Maag      EN0 := Signal Wert selektiert
//                               (S1 | S2 | S3)  AND ENABLE
//
//29.01.2013   S.Maag      Anzeige aktiver Kanal (DSP_CHANNEL)
//--------------------------------------------------------------------------------
//
//HINWEISE:
AUTHOR : 'S.Maag'
FAMILY : Maagic7
VERSION : 2.0


VAR_INPUT
  S1 : BOOL ;
  S2 : BOOL ;
  S3 : BOOL ;
  S4 : BOOL ;
  ENABLE : BOOL ;
  DINT1 : DINT ;
  DINT2 : DINT ;
  DINT3 : DINT ;
  DINT4 : DINT ;
END_VAR
VAR_OUTPUT
  DSP_CHANNEL : INT ;	//Displays the activated channel
END_VAR
BEGIN
NETWORK
TITLE =

      UN    #ENABLE; // keine Freigabe, dann 0 ausgeben
      SPB   STOP;

      U     #S1;
      SPB   S1;
      U     #S2;
      SPB   S2;
      U     #S3;
      SPB   S3;
      U     #S4;
      SPB   S4;

      SPA   STOP;

S1:   L     1; // Wert für Kanalanzeige
      L     #DINT1;
      SPA   SAVE;

S2:   L     2;
      L     #DINT2;
      SPA   SAVE;

S3:   L     3;
      L     #DINT3;
      SPA   SAVE;

S4:   L     4;
      L     #DINT4;
      SPA   SAVE;

STOP: CLR   ; // EN0-Ausgang =0, da Stopp
      L     0; // Wert für Kanalanzeige
      L     L#0; // Wert für Multiplexer

SAVE: SAVE  ;
      T     #RET_VAL; // Mulitplexer Ausgang
      TAK   ; // Wert aktiver Kanal
      T     #DSP_CHANNEL; // Anzeige aktiver Kanal

END_FUNCTION

FUNCTION "m7b_MAPx4xDINT" : VOID
TITLE =4x mapping for DOUBLE INTEGER
//This function maps 4 individual Inputs to 4 individual Outputs using the
//mapping table MAP_1..MAP_4. There is no check for double using an INPUT.
//
//OUT(1)=IN(MAP_1)
//OUT(2)=IN(MAP_2)
//OUT(3)=IN(MAP_3)
//OUT(4)=IN(MAP_4)
//
//AUTOR: Stefan Maag, Dipl.-Ing. (FH) Elektrotechnik
//DATUM: 07/2012
//
//AENDERUNGSVERMERKE:
//--------------------------------------------------------------------------------
//DATUM        NAME            AENDERUNG
//--------------------------------------------------------------------------------
//
//--------------------------------------------------------------------------------
//HINWEISE:
//Seit 07.04.2020 neue Version in SCL mit 2 mapping Modes.
//Für neue Projekte nur noch neue Version verwenden
AUTHOR : 'S.Maag'
FAMILY : Maagic7
VERSION : 0.1


VAR_INPUT
  IN_1 : DINT ;	//Input Value 1
  IN_2 : DINT ;	//Input Value 2
  IN_3 : DINT ;	//Input Value 3
  IN_4 : DINT ;	//Input Value 4
  ZERO_VAL : DINT ;	//Zero Value (used as 'zero', if no mapping)
  MAP_1 : INT ;	//Source Nr. for OUT_1: OUT_1=IN(MAP_1)
  MAP_2 : INT ;	//Source Nr. for OUT_2: OUT_2=IN(MAP_2)
  MAP_3 : INT ;	//Source Nr. for OUT_3: OUT_3=IN(MAP_3)
  MAP_4 : INT ;	//Source Nr. for OUT_4: OUT_3=IN(MAP_4)
END_VAR
VAR_OUTPUT
  OUT_1 : DINT ;
  OUT_2 : DINT ;
  OUT_3 : DINT ;
  OUT_4 : DINT ;
END_VAR
BEGIN
NETWORK
TITLE =

      SET   ;
      SAVE  ;
      CLR   ;

NETWORK
TITLE =MAP 1 : OUT_1 := IN (MAP_1)

      L     #MAP_1; // MAPPING-ZIEL Eingang 1
      SPL   a0; // Sprungziel bei MAP > 4
      SPA   a0; // MAP TO 0
      SPA   a1; // MAP TO 1
      SPA   a2; // MAP TO 2
      SPA   a3; // MAP TO 3
      SPA   a4; // MAO TO 4

a0:   L     #ZERO_VAL;
      SPA   aSAV;
a1:   L     #IN_1;
      SPA   aSAV;
a2:   L     #IN_2;
      SPA   aSAV;
a3:   L     #IN_3;
      SPA   aSAV;
a4:   L     #IN_4;
aSAV: T     #OUT_1;
NETWORK
TITLE =MAP 2 : OUT_2 := IN (MAP_2)

      L     #MAP_2; // MAPPING-ZIEL Eingang 2
      SPL   b0; // Sprungziel bei MAP > 4
      SPA   b0; // MAP TO 0
      SPA   b1; // MAP TO 1
      SPA   b2; // MAP TO 2
      SPA   b3; // MAP TO 3
      SPA   b4; // MAO TO 4

b0:   L     #ZERO_VAL;
      SPA   bSAV;
b1:   L     #IN_1;
      SPA   bSAV;
b2:   L     #IN_2;
      SPA   bSAV;
b3:   L     #IN_3;
      SPA   bSAV;
b4:   L     #IN_4;
bSAV: T     #OUT_2;
NETWORK
TITLE =MAP 3 : OUT_3 := IN (MAP_3)

      L     #MAP_3; // MAPPING-ZIEL Eingang 3
      SPL   c0; // Sprungziel bei MAP > 4
      SPA   c0; // MAP TO 0
      SPA   c1; // MAP TO 1
      SPA   c2; // MAP TO 2
      SPA   c3; // MAP TO 3
      SPA   c4; // MAO TO 4

c0:   L     #ZERO_VAL;
      SPA   cSAV;
c1:   L     #IN_1;
      SPA   cSAV;
c2:   L     #IN_2;
      SPA   cSAV;
c3:   L     #IN_3;
      SPA   cSAV;
c4:   L     #IN_4;
cSAV: T     #OUT_3;
NETWORK
TITLE =MAP 4 : OUT_4 := IN (MAP_4)

      L     #MAP_4; // MAPPING-ZIEL Eingang 4
      SPL   d0; // Sprungziel bei MAP > 4
      SPA   d0; // MAP TO 0
      SPA   d1; // MAP TO 1
      SPA   d2; // MAP TO 2
      SPA   d3; // MAP TO 3
      SPA   d4; // MAO TO 4

d0:   L     #ZERO_VAL;
      SPA   dSAV;
d1:   L     #IN_1;
      SPA   dSAV;
d2:   L     #IN_2;
      SPA   dSAV;
d3:   L     #IN_3;
      SPA   dSAV;
d4:   L     #IN_4;
dSAV: T     #OUT_4;
END_FUNCTION

FUNCTION "m7b_X_Switch_DINT" : VOID
TITLE =X_Switch_DINT : Kreuzschalter für DINT-Werte
//KREUZSCHALTUNG
//
//X_Switch : False: 1:1 - Schaltung OUT1:IN1; OUT2=IN2
//           True :   X - Schaltung OUT1:IN2; OUT2=IN1
//
//IN1 : Eingang 1
//IN2 : Eingang 2
//OUT1: Ausgang 1
//OUT2: Ausgang 2
//
//FC-ENO : Der X_Switch Eingang wird auf ENO druchgeschleift
//
//AUTOR: Stefan Maag, Dipl.-Ing. (FH) Elektrotechnik
//DATUM: 03/2009
//INTERNET: www.maagic7.de
//
//AENDERUNGSVERMERKE:
//--------------------------------------------------------------------------------
//DATUM        NAME            AENDERUNG
//--------------------------------------------------------------------------------
//
//--------------------------------------------------------------------------------
//
//HINWEISE:
AUTHOR : 'S.Maag'
FAMILY : Maagic7
VERSION : 0.1


VAR_INPUT
  X_Switch : BOOL ;	//False: 1:1 Schaltung; True: X-Schaltung
  IN1 : DINT ;	//Eingangswert 1
  IN2 : DINT ;	//Eingangswert 2
END_VAR
VAR_OUTPUT
  OUT1 : DINT ;
  OUT2 : DINT ;
END_VAR
BEGIN
NETWORK
TITLE =Kreuschalterfunktion

      U     #X_Switch; // Wenn Kreuzschaltung aktiv
      SAVE  ; // Schalter auf ENO durchschleifen
      SPB   X; // Ausgänge kreuz geschaltet

      L     #IN1; // Ausgänge 1:1 schalten
      T     #OUT1;

      L     #IN2;
      T     #OUT2;
      BEA   ;

X:    L     #IN1; // Ausgänge über Kreuz schalten
      T     #OUT2;

      L     #IN2;
      T     #OUT1;



END_FUNCTION

FUNCTION "m7b_InvertRange_DINT" : DINT
TITLE =InvertRange_DINT: Invertiert einen Bereich (Messrichtungsumkehr)
//Invertiert einen Wertebereich (Messrichtungsumkehr), vertauscht sozusagen Ober-
//und Untergrenze.
//Bei symetrischen Wertebereichen: MIN = -MAX ist das einfach eine
//Vorzeichenumkehr.
//
//ENO : Übersteuerungsanzeige: der invertierte Wert liegt ausserhalb des
//      Wertebereichs. Dieses Signal kann z.B. dazu verwendet werden um
//      eine gesonderte verarbeitung im Fehlerfalle druchzuführen.
//
//
//z.B. MIN=-100 MAX=100 VALUE=20 : Xinv= -20
//     MIN=  20 MAX=100 VALUE=20 : Xinv= 100
//                      VALUE=50 : Xinv=  70
//
//Xinv= MIN + MAX - VALUE
//
//
//AUTOR: Stefan Maag, Dipl.-Ing. (FH) Elektrotechnik
//DATUM: 10/2008
//INTERNET: www.maagic7.de
//
//AENDERUNGSVERMERKE:
//--------------------------------------------------------------------------------
//DATUM        NAME            AENDERUNG
//--------------------------------------------------------------------------------
//
//--------------------------------------------------------------------------------
//
//HINWEISE:
AUTHOR : 'S.Maag'
FAMILY : Maagic7
VERSION : 0.1


VAR_INPUT
  VALUE : DINT ;	//Value to invert
  MIN : DINT ;	//Minimum of Range
  MAX : DINT ;	//Maximum of Range
END_VAR
BEGIN
NETWORK
TITLE =Invert Range: Wertebereich umkehren
//Xinv= MAX - VALUE + MIN  :  Bessere Berechnung wegen Überläufen
      L     #MAX;
      L     #VALUE;
      -D    ;
      L     #MIN;
      +D    ;
      T     #RET_VAL;
NETWORK
TITLE =FC-ENO-Ausgang als Übersteuerungsanzeige

      L     #MAX; // Maximalwert
      >D    ; // Wert > MAX
      SPB   SAVE; // Max-Wert überschritten
      TAK   ; // Ausgangswert in Akku 1 zurueck
      L     #MIN;
      <D    ;
      SPB   SAVE; // MinWert unterschritten
      CLR   ;
SAVE: SAVE  ;
      CLR   ;
END_FUNCTION

FUNCTION "m7b_MinDiffABS_DINT" : VOID
TITLE =MinDiffABS_DINT: Minimale Absolutdifferenz 2er DINT-Werte ok!
//Überprüft, ob die absolute Differenz (absolut) zweier DINT dem angebegenen
//Mindestwert entspricht. Wenn ja, dann wird ENO=True
//
//BENÖTIGTE SFCs: keine
//
//AUTOR: Stefan Maag, Dipl.-Ing. (FH) Elektrotechnik
//DATUM: 8/2008
//INTERNET: www.maagic7.de
//
//AENDERUNGSVERMERKE:
//--------------------------------------------------------------------------------
//DATUM        NAME        AENDERUNG
//--------------------------------------------------------------------------------
//10.09.2020   S.Maag      Ausgang dDiff hinzugefügt
//--------------------------------------------------------------------------------
//
//HINWEISE:
AUTHOR : 'S.Maag'
FAMILY : Maagic7
VERSION : 0.1


VAR_INPUT
  VAL_1 : DINT ;
  VAL_2 : DINT ;
  MinDiff : DINT ;
END_VAR
VAR_OUTPUT
  dDiff : DINT ;	//Differenz=ABS(VAL_1-VAL_2)
END_VAR
VAR_TEMP
  aktSysTime : TIME ;	//aktuelle Systemzeit
END_VAR
BEGIN
NETWORK
TITLE =prüfen ob Differenz ok

      L     #VAL_1;
      L     #VAL_2;
      -D    ;
      SPP   pos;
      NEGD  ;
pos:  T     #dDiff;
      L     #MinDiff;
      >=D   ;
      SAVE  ;

END_FUNCTION

FUNCTION "m7b_SchleppZeiger_DINT" : VOID
TITLE =SchleppZeiger_DINT: Schleppzeiger für DINT (drag indicator)
//Schleppzeiger für Doppel-Integerwerte
//
//Der FC-ENO-Ausgang wird dann "1", wenn der Schleppzeiger einen neuen Wert
//erhält, ansonsten ist der FC-ENO-Ausgang "0"
//
//AUTOR: Stefan Maag, Dipl.-Ing. (FH) Elektrotechnik
//DATUM: 9/2004
//INTERNET: www.maagic7.de
//
//AENDERUNGSVERMERKE:
//--------------------------------------------------------------------------------
//DATUM        NAME            AENDERUNG
//--------------------------------------------------------------------------------
//
//--------------------------------------------------------------------------------
//
//HINWEISE:
AUTHOR : 'S.Maag'
FAMILY : Maagic7
VERSION : 0.1


VAR_INPUT
  dValue : DINT ;	//aktueller Wert
  cfgMinMax : BOOL ;	//Konfig.: 0=Minimum Schleppzeiger 1=Maximum Schleppzeiger
  Init : BOOL ;	//Initialisierung, Schleppzeiger wird auf aktuellen Wert gesetzt
END_VAR
VAR_IN_OUT
  SchleppZeiger : DINT ;	//Schleppzeiger-Wert
END_VAR
BEGIN
NETWORK
TITLE =

      U     #Init;
      SPB   INIT;

      U     #cfgMinMax; // Maximum Schleppzeiger
      SPB   MAX;

      L     #SchleppZeiger; // Minimum Schleppzeiger
      L     #dValue;
      <D    ;
      SPB   END;
      SPA   SAVE;

INIT: L     #dValue; // Schleppzeicher initialisieren
      SPA   SAVE;

MAX:  L     #SchleppZeiger;
      L     #dValue;
      >D    ;
      SPB   END;

SAVE: T     #SchleppZeiger;
      SET   ;
      SAVE  ;
      CLR   ;
      BEA   ;

END:  CLR   ;
      SAVE  ;

END_FUNCTION

FUNCTION "m7b_ChangeEvent_REAL" : VOID
TITLE =Ereignis REAL Wert hat sich geändert
//Der FC-ENO-Ausgang wird für einen Zyklus "1", wenn der sich der Eingangswert
//geändert hat, ansonsten ist der FC-ENO-Ausgang "0"
//
//AUTOR: Stefan Maag, Dipl.-Ing. (FH) Elektrotechnik
//DATUM: 8/2008
//INTERNET: www.maagic7.de
//
//AENDERUNGSVERMERKE:
//--------------------------------------------------------------------------------
//DATUM        NAME            AENDERUNG
//--------------------------------------------------------------------------------
//
//--------------------------------------------------------------------------------
//
//HINWEISE:
AUTHOR : 'S.Maag'
FAMILY : Maagic7
VERSION : 0.1


VAR_INPUT
  inREAL : REAL ;
END_VAR
VAR_IN_OUT
  memREAL : REAL ;
END_VAR
BEGIN
NETWORK
TITLE =

      L     #inREAL; // Eingangwert
      L     #memREAL; // letzter Wert
      <>R   ; // ungleich!
      SAVE  ; // als ENO ausgeben
      SPB   do; // und neuen
      BEA   ;
do:   L     #inREAL; // Wert speichern
      T     #memREAL;

END_FUNCTION

FUNCTION "m7b_RP_WRITE_REAL" : VOID
TITLE =Ringpuffer schreiben REAL-Werte
//AUTOR: Stefan Maag, Dipl.-Ing. (FH) Elektrotechnik
//DATUM: 7/2008
//INTERNET: www.maagic7.de
//
//AENDERUNGSVERMERKE:
//--------------------------------------------------------------------------------
//DATUM        NAME        AENDERUNG
//--------------------------------------------------------------------------------
//09.07.2010   S.Maag      ENO nur True, wenn Ringpuffer geschrieben/verarbeitet
//                         wird, sonst FALSE
//--------------------------------------------------------------------------------
//
//HINWEISE:
AUTHOR : 'S.Maag'
FAMILY : Maagic7
VERSION : 0.1


VAR_INPUT
  DB_RP : BLOCK_DB ;
  RP_POS : BOOL ;	//Ringpuffer schreiben positiv
  RP_NEG : BOOL ;	//Ringpuffer schreiben negativ
  IN_REAL : DINT ;	//Eingangswert DINT
END_VAR
VAR_IN_OUT
  RP_IDX : INT ;	//Indexwert Ringpuffer 0..255
END_VAR
VAR_TEMP
  AR1 : DWORD ;
END_VAR
BEGIN
NETWORK
TITLE =

      TAR1  #AR1; // Adressregister 1 sichern

NETWORK
TITLE =

      U     #RP_POS; // positiver Impuls := Ringpuffer vorwärts
      SPB   pos;

      U     #RP_NEG; // negativer Impuls := Ringpuffer rückwärts
      SPB   neg;

      CLR   ; // ENO = FALSE, => keine Verarbeitung
      SAVE  ;
      BEA   ;

pos:  L     #RP_IDX; // positiver Impuls := Ringpuffer vorwärts
      INC   1; // INC: Bytebefehl 0..255
      SPA   save;

neg:  L     #RP_IDX; // negativer Impuls := Ringpuffer rückwärts
      DEC   1; // DEC: Bytebefehl 0..255

save: T     #RP_IDX; // Indexwert Ringpuffer 0..255
      SLD   5; // SLD 2 wegen DINT-Werten=>Byte + SLD 3 wegen Pointer
      L     P#0.0; // 0-Pointer addieren
      +D    ; // Pointer auf Daten erzeugen
      LAR1  ; // in Adressregister 1 laden

      AUF   #DB_RP; // Ringpuffer DB öffnen
      L     #IN_REAL; // Eingangswert laden
      T     DBD [AR1,P#0.0]; // in DB speichern

      LAR1  #AR1; // ursprüngliches Adressregister 1 herstellen
      SET   ; // ENO = TRUE, => Verarbeitung
      SAVE  ;
      BEA   ;


END_FUNCTION

FUNCTION "m7b_RP_READ_REAL" : REAL
TITLE =Ringpuffer lesen REAL-Werte
//AUTOR: Stefan Maag, Dipl.-Ing. (FH) Elektrotechnik
//DATUM: 7/2008
//INTERNET: www.maagic7.de
//
//AENDERUNGSVERMERKE:
//--------------------------------------------------------------------------------
//DATUM        NAME        AENDERUNG
//--------------------------------------------------------------------------------
//
//--------------------------------------------------------------------------------
//
//HINWEISE:
AUTHOR : 'S.Maag'
FAMILY : Maagic7
VERSION : 0.1


VAR_INPUT
  DB_RP : BLOCK_DB ;
  RP_IDX : INT ;	//Ringpuffer Index
  RP_OFFSET : INT ;	//Offeset Ringpufferindex
END_VAR
VAR_TEMP
  AR1 : DWORD ;
END_VAR
BEGIN
NETWORK
TITLE =

      TAR1  #AR1; // Adressregister 1 sichern

      L     #RP_IDX; // aktueller Ringpuffer-Index
      L     #RP_OFFSET; // Offset für lesen
      -I    ;
      L     W#16#FF; // auf 0..255 begrenzen
      UW    ;
      SLD   5; // SLD 2 wegen DINT-Werten=>Byte + SLD 3 wegen Pointer
      L     P#0.0; // 0-Pointer addieren
      +D    ; // Pointer auf Daten erzeugen
      LAR1  ; // in Adressregister 1 laden

      AUF   #DB_RP; // Ringpuffer DB öffnen
      L     DBD [AR1,P#0.0]; // Wert aus Ringpuffer laden
      T     #RET_VAL; // Rückgabewert

      LAR1  #AR1; // ursprüngliches Adressregister 1 herstellen
      SET   ;
      SAVE  ;
      CLR   ;

END_FUNCTION

FUNCTION_BLOCK "m7b_CYCLE_TIME_SPLITTER"
TITLE =Zykluszeitverteilung
AUTHOR : 'S.Maag'
FAMILY : Maagic7
VERSION : 0.1


VAR_INPUT
  RESET : BOOL ;
END_VAR
VAR_OUTPUT
  CYC_1of2 : BOOL ;
  CYC_2of2 : BOOL ;
  CYC_1of4 : BOOL ;
  CYC_2of4 : BOOL ;
  CYC_3of4 : BOOL ;
  CYC_4of4 : BOOL ;
END_VAR
VAR
  mem_1Of4 : BOOL ;
END_VAR
BEGIN
NETWORK
TITLE =



NETWORK
TITLE =Zyklus 1 von 2
//======================================================================
//                    C Y C L E   1 o f 2
//======================================================================
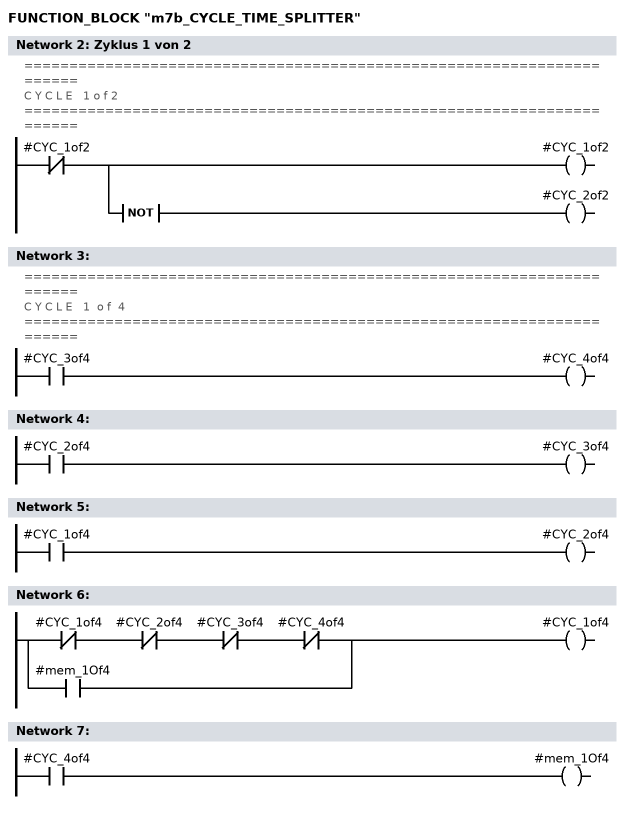
      UN    #CYC_1of2;
      =     L      0.0;
      U     L      0.0;
      BLD   102;
      =     #CYC_1of2;
      U     L      0.0;
      NOT   ;
      =     #CYC_2of2;
NETWORK
TITLE =
//======================================================================
//                    C Y C L E   1  o f  4
//======================================================================
      U     #CYC_3of4;
      =     #CYC_4of4;
NETWORK
TITLE =

      U     #CYC_2of4;
      =     #CYC_3of4;
NETWORK
TITLE =

      U     #CYC_1of4;
      =     #CYC_2of4;
NETWORK
TITLE =

      UN    #CYC_1of4;
      UN    #CYC_2of4;
      UN    #CYC_3of4;
      UN    #CYC_4of4;
      O     #mem_1Of4;
      =     #CYC_1of4;
NETWORK
TITLE =

      U     #CYC_4of4;
      =     #mem_1Of4;
NETWORK
TITLE =

      U     BIE;
      UN    #RESET;
      SAVE  ;
      BEB   ;
NETWORK
TITLE =

      U     #RESET;
      R     #CYC_1of2;
      R     #CYC_2of2;
      R     #CYC_1of4;
      R     #CYC_2of4;
      R     #CYC_3of4;
      R     #CYC_4of4;
END_FUNCTION_BLOCK

FUNCTION "m7b_MUXx3xREAL" : REAL
TITLE =3-fach REAL Multiplexer
//AUTOR: Stefan Maag, Dipl.-Ing. (FH) Elektrotechnik
//DATUM: 8/2008
//INTERNET: www.maagic7.de
//
//AENDERUNGSVERMERKE:
//--------------------------------------------------------------------------------
//DATUM        NAME        AENDERUNG
//--------------------------------------------------------------------------------
//25.08.2008   S.Maag      enstanden aus MUXx3xINT
//
//24.04.2009   S.Maag      EN0 := Signal Wert selektiert
//                               (S1 | S2 | S3)  AND ENABLE
//
//29.01.2013   S.Maag      Anzeige aktiver Kanal (DSP_CHANNEL)
//--------------------------------------------------------------------------------
//
//HINWEISE:
AUTHOR : 'S.Maag'
FAMILY : Maagic7
VERSION : 2.0


VAR_INPUT
  S1 : BOOL ;
  S2 : BOOL ;
  S3 : BOOL ;
  ENABLE : BOOL ;
  REAL1 : REAL ;
  REAL2 : REAL ;
  REAL3 : REAL ;
END_VAR
VAR_OUTPUT
  DSP_CHANNEL : INT ;	//Displays the activated channel
END_VAR
BEGIN
NETWORK
TITLE =

      UN    #ENABLE; // keine Freigabe, dann 0 ausgeben
      SPB   STOP;

      U     #S1;
      SPB   S1;
      U     #S2;
      SPB   S2;
      U     #S3;
      SPB   S3;

      SPA   STOP;

S1:   L     1; // Wert für Kanalanzeige
      L     #REAL1;
      SPA   SAVE;

S2:   L     2;
      L     #REAL2;
      SPA   SAVE;

S3:   L     3;
      L     #REAL3;
      SPA   SAVE;

STOP: CLR   ; // EN0-Ausgang =0, da Stopp
      L     0; // Wert für Kanalanzeige
      L     0.000000e+000; // Wert für Multiplexer

SAVE: SAVE  ;
      T     #RET_VAL; // Mulitplexer Ausgang
      TAK   ; // Wert aktiver Kanal
      T     #DSP_CHANNEL; // Anzeige aktiver Kanal

END_FUNCTION

FUNCTION "m7b_MUXx4xREAL" : REAL
TITLE =4-fach REAL Multiplexer
//AUTOR: Stefan Maag, Dipl.-Ing. (FH) Elektrotechnik
//DATUM: 8/2008
//INTERNET: www.maagic7.de
//
//AENDERUNGSVERMERKE:
//--------------------------------------------------------------------------------
//DATUM        NAME        AENDERUNG
//--------------------------------------------------------------------------------
//25.08.2008   S.Maag      enstanden aus MUXx3xINT
//
//24.04.2009   S.Maag      EN0 := Signal Wert selektiert
//                               (S1 | S2 | S3)  AND ENABLE
//--------------------------------------------------------------------------------
//
//HINWEISE:
AUTHOR : 'S.Maag'
FAMILY : Maagic7
VERSION : 2.0


VAR_INPUT
  S1 : BOOL ;
  S2 : BOOL ;
  S3 : BOOL ;
  S4 : BOOL ;
  ENABLE : BOOL ;
  REAL1 : REAL ;
  REAL2 : REAL ;
  REAL3 : REAL ;
  REAL4 : REAL ;
END_VAR
VAR_OUTPUT
  DSP_CHANNEL : INT ;	//Displays the activated channel
END_VAR
BEGIN
NETWORK
TITLE =

      UN    #ENABLE; // keine Freigabe, dann 0 ausgeben
      SPB   STOP;

      U     #S1;
      SPB   S1;
      U     #S2;
      SPB   S2;
      U     #S3;
      SPB   S3;
      U     #S4;
      SPB   S4;

      SPA   STOP;

S1:   L     1; // Wert für Kanalanzeige
      L     #REAL1;
      SPA   SAVE;

S2:   L     2;
      L     #REAL2;
      SPA   SAVE;

S3:   L     3;
      L     #REAL3;
      SPA   SAVE;

S4:   L     4;
      L     #REAL4;
      SPA   SAVE;

STOP: CLR   ; // EN0-Ausgang =0, da Stopp
      L     0; // Wert für Kanalanzeige
      L     0.000000e+000; // Wert für Multiplexer

SAVE: SAVE  ;
      T     #RET_VAL; // Mulitplexer Ausgang
      TAK   ; // Wert aktiver Kanal
      T     #DSP_CHANNEL; // Anzeige aktiver Kanal

END_FUNCTION

FUNCTION "m7b_MAPx4xREAL" : VOID
TITLE =4x mapping for REAL
//This function maps 4 individual Inputs to 4 individual Outputs using the
//mapping table MAP_1..MAP_4. There is no check for double using an INPUT.
//
//OUT(1)=IN(MAP_1)
//OUT(2)=IN(MAP_2)
//OUT(3)=IN(MAP_3)
//OUT(4)=IN(MAP_4)
//
//AUTOR: Stefan Maag, Dipl.-Ing. (FH) Elektrotechnik
//DATUM: 07/2012
//
//AENDERUNGSVERMERKE:
//--------------------------------------------------------------------------------
//DATUM        NAME            AENDERUNG
//--------------------------------------------------------------------------------
//
//--------------------------------------------------------------------------------
//HINWEISE:
//Seit 07.04.2020 neue Version in SCL mit 2 mapping Modes.
//Für neue Projekte nur noch neue Version verwenden
AUTHOR : 'S.Maag'
FAMILY : Maagic7
VERSION : 0.1


VAR_INPUT
  IN_1 : REAL ;	//Input Value 1
  IN_2 : REAL ;	//Input Value 2
  IN_3 : REAL ;	//Input Value 3
  IN_4 : REAL ;	//Input Value 4
  ZERO_VAL : REAL ;	//Zero Value (used as 'zero', if no mapping)
  MAP_1 : INT ;	//Source Nr. for OUT_1: OUT_1=IN(MAP_1)
  MAP_2 : INT ;	//Source Nr. for OUT_2: OUT_2=IN(MAP_2)
  MAP_3 : INT ;	//Source Nr. for OUT_3: OUT_3=IN(MAP_3)
  MAP_4 : INT ;	//Source Nr. for OUT_4: OUT_3=IN(MAP_4)
END_VAR
VAR_OUTPUT
  OUT_1 : REAL ;
  OUT_2 : REAL ;
  OUT_3 : REAL ;
  OUT_4 : REAL ;
END_VAR
BEGIN
NETWORK
TITLE =

      SET   ;
      SAVE  ;
      CLR   ;

NETWORK
TITLE =MAP 1 : OUT_1 := IN (MAP_1)

      L     #MAP_1; // MAPPING-ZIEL Eingang 1
      SPL   a0; // Sprungziel bei MAP > 4
      SPA   a0; // MAP TO 0
      SPA   a1; // MAP TO 1
      SPA   a2; // MAP TO 2
      SPA   a3; // MAP TO 3
      SPA   a4; // MAO TO 4

a0:   L     #ZERO_VAL;
      SPA   aSAV;
a1:   L     #IN_1;
      SPA   aSAV;
a2:   L     #IN_2;
      SPA   aSAV;
a3:   L     #IN_3;
      SPA   aSAV;
a4:   L     #IN_4;
aSAV: T     #OUT_1;
NETWORK
TITLE =MAP 2 : OUT_2 := IN (MAP_2)

      L     #MAP_2; // MAPPING-ZIEL Eingang 2
      SPL   b0; // Sprungziel bei MAP > 4
      SPA   b0; // MAP TO 0
      SPA   b1; // MAP TO 1
      SPA   b2; // MAP TO 2
      SPA   b3; // MAP TO 3
      SPA   b4; // MAO TO 4

b0:   L     #ZERO_VAL;
      SPA   bSAV;
b1:   L     #IN_1;
      SPA   bSAV;
b2:   L     #IN_2;
      SPA   bSAV;
b3:   L     #IN_3;
      SPA   bSAV;
b4:   L     #IN_4;
bSAV: T     #OUT_2;
NETWORK
TITLE =MAP 3 : OUT_3 := IN (MAP_3)

      L     #MAP_3; // MAPPING-ZIEL Eingang 3
      SPL   c0; // Sprungziel bei MAP > 4
      SPA   c0; // MAP TO 0
      SPA   c1; // MAP TO 1
      SPA   c2; // MAP TO 2
      SPA   c3; // MAP TO 3
      SPA   c4; // MAO TO 4

c0:   L     #ZERO_VAL;
      SPA   cSAV;
c1:   L     #IN_1;
      SPA   cSAV;
c2:   L     #IN_2;
      SPA   cSAV;
c3:   L     #IN_3;
      SPA   cSAV;
c4:   L     #IN_4;
cSAV: T     #OUT_3;
NETWORK
TITLE =MAP 4 : OUT_4 := IN (MAP_4)

      L     #MAP_4; // MAPPING-ZIEL Eingang 4
      SPL   d0; // Sprungziel bei MAP > 4
      SPA   d0; // MAP TO 0
      SPA   d1; // MAP TO 1
      SPA   d2; // MAP TO 2
      SPA   d3; // MAP TO 3
      SPA   d4; // MAO TO 4

d0:   L     #ZERO_VAL;
      SPA   dSAV;
d1:   L     #IN_1;
      SPA   dSAV;
d2:   L     #IN_2;
      SPA   dSAV;
d3:   L     #IN_3;
      SPA   dSAV;
d4:   L     #IN_4;
dSAV: T     #OUT_4;
END_FUNCTION

FUNCTION "m7b_X_Switch_REAL" : VOID
TITLE =X_Switch_DINT : Kreuzschalter für REAL-Werte
//KREUZSCHALTUNG
//
//X_Switch : False: 1:1 - Schaltung OUT1:IN1; OUT2=IN2
//           True :   X - Schaltung OUT1:IN2; OUT2=IN1
//
//IN1 : Eingang 1
//IN2 : Eingang 2
//OUT1: Ausgang 1
//OUT2: Ausgang 2
//
//FC-ENO : Der X_Switch Eingang wird auf ENO druchgeschleift
//
//AUTOR: Stefan Maag, Dipl.-Ing. (FH) Elektrotechnik
//DATUM: 03/2009
//INTERNET: www.maagic7.de
//
//AENDERUNGSVERMERKE:
//--------------------------------------------------------------------------------
//DATUM        NAME            AENDERUNG
//--------------------------------------------------------------------------------
//
//--------------------------------------------------------------------------------
//
//HINWEISE:
AUTHOR : 'S.Maag'
FAMILY : Maagic7
VERSION : 0.1


VAR_INPUT
  X_Switch : BOOL ;	//False: 1:1 Schaltung; True: X-Schaltung
  IN1 : REAL ;	//Eingangswert 1
  IN2 : REAL ;	//Eingangswert 2
END_VAR
VAR_OUTPUT
  OUT1 : REAL ;
  OUT2 : REAL ;
END_VAR
BEGIN
NETWORK
TITLE =Kreuschalterfunktion

      U     #X_Switch; // Wenn Kreuzschaltung aktiv
      SAVE  ; // Schalter auf ENO durchschleifen
      SPB   X; // Ausgänge kreuz geschaltet

      L     #IN1; // Ausgänge 1:1 schalten
      T     #OUT1;

      L     #IN2;
      T     #OUT2;
      BEA   ;

X:    L     #IN1; // Ausgänge über Kreuz schalten
      T     #OUT2;

      L     #IN2;
      T     #OUT1;



END_FUNCTION

FUNCTION "m7b_InvertRange_REAL" : REAL
TITLE =InvertRange_REAL: Invertiert einen Bereich (Messrichtungsumkehr)
//Invertiert einen Wertebereich (Messrichtungsumkehr), vertauscht sozusagen Ober-
//und Untergrenze.
//Bei symetrischen Wertebereichen: MIN = -MAX ist das einfach eine
//Vorzeichenumkehr.
//
//ENO : Übersteuerungsanzeige: der invertierte Wert liegt ausserhalb des
//      Wertebereichs. Dieses Signal kann z.B. dazu verwendet werden um
//      eine gesonderte verarbeitung im Fehlerfalle druchzuführen.
//
//
//z.B. MIN=-100 MAX=100 VALUE=20 : Xinv= -20
//     MIN=  20 MAX=100 VALUE=20 : Xinv= 100
//                      VALUE=50 : Xinv=  70
//
//Xinv= MIN + MAX - VALUE
//
//
//AUTOR: Stefan Maag, Dipl.-Ing. (FH) Elektrotechnik
//DATUM: 10/2008
//INTERNET: www.maagic7.de
//
//AENDERUNGSVERMERKE:
//--------------------------------------------------------------------------------
//DATUM        NAME            AENDERUNG
//--------------------------------------------------------------------------------
//
//--------------------------------------------------------------------------------
//
//HINWEISE:
AUTHOR : 'S.Maag'
FAMILY : Maagic7
VERSION : 0.1


VAR_INPUT
  VALUE : REAL ;	//Value to invert
  MIN : REAL ;	//Minimum of Range
  MAX : REAL ;	//Maximum of Range
END_VAR
BEGIN
NETWORK
TITLE =Invert Range: Wertebereich umkehren
//Xinv= MAX - VALUE + MIN  :  Bessere Berechnung wegen Überläufen
      L     #MAX;
      L     #VALUE;
      -R    ;
      L     #MIN;
      +R    ;
      T     #RET_VAL;
NETWORK
TITLE =FC-ENO-Ausgang als Übersteuerungsanzeige

      L     #MAX; // Maximalwert
      >R    ; // Wert > MAX
      SPB   SAVE; // Max-Wert überschritten
      TAK   ; // Ausgangswert in Akku 1 zurueck
      L     #MIN;
      <R    ;
      SPB   SAVE; // MinWert unterschritten
      CLR   ;
SAVE: SAVE  ;
      CLR   ;
END_FUNCTION

FUNCTION "m7b_MinDiffABS_REAL" : VOID
TITLE =MinDiffABS_REAL: Minimale Absolutdifferenz 2er REAL-Werte ok!
//Überprüft, ob die absolute Differenz (absolut) zweier DINT dem angebegenen
//Mindestwert entspricht. Wenn ja, dann wird ENO=True
//
//BENÖTIGTE SFCs: keine
//
//AUTOR: Stefan Maag, Dipl.-Ing. (FH) Elektrotechnik
//DATUM: 8/2008
//INTERNET: www.maagic7.de
//
//AENDERUNGSVERMERKE:
//--------------------------------------------------------------------------------
//DATUM        NAME        AENDERUNG
//--------------------------------------------------------------------------------
//--------------------------------------------------------------------------------
//10.09.2020   S.Maag      Ausgang rDiff hinzugefügt
//--------------------------------------------------------------------------------
//
//HINWEISE:
AUTHOR : 'S.Maag'
FAMILY : Maagic7
VERSION : 0.1


VAR_INPUT
  VAL_1 : REAL ;
  VAL_2 : REAL ;
  MinDiff : REAL ;
END_VAR
VAR_OUTPUT
  rDiff : REAL ;	//Differenz=ABS(VAL_1-VAL_
END_VAR
VAR_TEMP
  aktSysTime : TIME ;	//aktuelle Systemzeit
END_VAR
BEGIN
NETWORK
TITLE =prüfen ob Differenz ok

      L     #VAL_1;
      L     #VAL_2;
      -R    ;
      SPP   pos;
      NEGR  ;
pos:  T     #rDiff;
      L     #MinDiff;
      >=R   ;
      SAVE  ;

END_FUNCTION

FUNCTION "m7b_SchleppZeiger_REAL" : VOID
TITLE =SchleppZeiger_REAL: Schleppzeiger für REAL
//Schleppzeiger für REAL-Werte
//
//Der FC-ENO-Ausgang wird dann "1", wenn der Schleppzeiger einen neuen Wert
//erhält, ansonsten ist der FC-ENO-Ausgang "0"
//
//AUTOR: Stefan Maag, Dipl.-Ing. (FH) Elektrotechnik
//DATUM: 9/2004
//INTERNET: www.maagic7.de
//
//AENDERUNGSVERMERKE:
//--------------------------------------------------------------------------------
//DATUM        NAME            AENDERUNG
//--------------------------------------------------------------------------------
//
//--------------------------------------------------------------------------------
//
//HINWEISE:
AUTHOR : 'S.Maag'
FAMILY : Maagic7
VERSION : 0.1


VAR_INPUT
  rValue : REAL ;	//aktueller Wert
  cfgMinMax : BOOL ;	//Konfig.: 0=Minimum Schleppzeiger 1=Maximum Schleppzeiger
  Init : BOOL ;	//Initialisierung, Schleppzeiger wird auf aktuellen Wert gesetzt
END_VAR
VAR_IN_OUT
  SchleppZeiger : REAL ;	//Schleppzeiger-Wert
END_VAR
BEGIN
NETWORK
TITLE =

      U     #Init;
      SPB   INIT;

      U     #cfgMinMax; // Maximum Schleppzeiger
      SPB   MAX;

      L     #SchleppZeiger; // Minimum Schleppzeiger
      L     #rValue;
      <R    ;
      SPB   END;
      SPA   SAVE;

INIT: L     #rValue; // Schleppzeicher initialisieren
      SPA   SAVE;

MAX:  L     #SchleppZeiger;
      L     #rValue;
      >R    ;
      SPB   END;

SAVE: T     #SchleppZeiger;
      SET   ;
      SAVE  ;
      CLR   ;
      BEA   ;

END:  CLR   ;
      SAVE  ;

END_FUNCTION

FUNCTION "m7b_ChangeEvent_TIME" : VOID
TITLE =Ereignis TIME Wert hat sich geändert
//Der FC-ENO-Ausgang wird für einen Zyklus "1", wenn der sich der Eingangswert
//geändert hat, ansonsten ist der FC-ENO-Ausgang "0"
//
//AUTOR: Stefan Maag, Dipl.-Ing. (FH) Elektrotechnik
//DATUM: 10/2008
//INTERNET: www.maagic7.de
//
//AENDERUNGSVERMERKE:
//--------------------------------------------------------------------------------
//DATUM        NAME            AENDERUNG
//--------------------------------------------------------------------------------
//
//--------------------------------------------------------------------------------
//
//HINWEISE:
AUTHOR : 'S.Maag'
FAMILY : Maagic7
VERSION : 0.1


VAR_INPUT
  inTIME : TIME ;
END_VAR
VAR_IN_OUT
  memTIME : TIME ;
END_VAR
BEGIN
NETWORK
TITLE =

      L     #inTIME; // Eingangwert
      L     #memTIME; // letzter Wert
      <>D   ; // ungleich!
      SAVE  ; // als ENO ausgeben
      SPB   do; // und neuen
      BEA   ;
do:   L     #inTIME; // Wert speichern
      T     #memTIME;

END_FUNCTION

FUNCTION "m7b_MinMaxLimit_TIME" : VOID
TITLE =Min/Max Begrenzung TIME; Begrenzungsanzeige im BIE-Bit / FC-ENO
//Min- Max- Begrenzung für TIME mit Begrenzungsanzeige
//
//BIE bzw. FC-ENO : 0 = Wert war ok       : Begrenzung nicht aktiv
//                  1 = Wert war nicht ok.: Begrenzung aktiv
//
//AUTOR: Stefan Maag, Dipl.-Ing. (FH) Elektrotechnik
//DATUM: 10/2008
//INTERNET: www.maagic7.de
//
//VERWENDUNG:
//Begrenzung eines Wertes auf den Min- Max- Bereich bei gleichzeitiger
//Weiterverarbeitung des Begrenzungssignals am FC-ENO-Ausgang z.B. zur Warn- bzw.
//Störungsanzeige oder zur direkten Weiterverschaltung.
//
//AENDERUNGSVERMERKE:
//--------------------------------------------------------------------------------
//DATUM        NAME            AENDERUNG
//--------------------------------------------------------------------------------
//
//--------------------------------------------------------------------------------
//
//HINWEISE:
AUTHOR : 'S.Maag'
FAMILY : Maagic7
VERSION : 0.1


VAR_INPUT
  min : TIME ;	//minimal Wert
  max : TIME ;	//maximal Wert
END_VAR
VAR_IN_OUT
  VALUE : TIME ;	//Sollwert
END_VAR
BEGIN
NETWORK
TITLE =MIN <= VALUE <= MAX

      L     #VALUE; // Sollwert
      L     #min; // minimal Wert
      <D    ;
      SPB   LIM; // Limitierung wenn VALUE < MIN
      TAK   ; // VALUE wieder in Akku 1
      L     #max; // Maximalwert
      >D    ;
      SPB   LIM; // Limitierung wenn VALUE > MAX

      CLR   ; // VKE löschen, da keine Begrenzung erfolgte
      SAVE  ; // BIE-Bit = 0, da Wert im Bereich war; ="Keine Begrenzung"
      BEA   ;

LIM:  T     #VALUE; // max.Wert als Sollwert ausgeben
      SET   ;
      SAVE  ; // VKE->BIE (=1=): Anzeige FC-ENO Ausgang (=Begrenzung)
      CLR   ;

END_FUNCTION

FUNCTION "m7b_BitToTIME" : VOID
TITLE =Bit To Time
//Je nach dem Wert des Eingangsbits wird der Wert
//VAL_0 oder VAL_1 als Ausgangswert VAL ausgegeben.
//Der Wert der Eingangsbits wird auf den FC-ENO-Ausgang durchgeschleift
//
//AUTOR: Stefan Maag, Dipl.-Ing. (FH) Elektrotechnik
//DATUM: 10/2008
//
//AENDERUNGSVERMERKE:
//--------------------------------------------------------------------------------
//DATUM        NAME            AENDERUNG
//--------------------------------------------------------------------------------
//
//--------------------------------------------------------------------------------
//
//HINWEISE:
AUTHOR : 'S.Maag'
FAMILY : Maagic7
VERSION : 0.1


VAR_INPUT
  BIT : BOOL ;
  VAL_0 : TIME ;
  VAL_1 : TIME ;
END_VAR
VAR_OUTPUT
  VAL : TIME ;
END_VAR
BEGIN
NETWORK
TITLE =

      U     #BIT;
      SAVE  ; // Wert von Bit auf FC-EN0
      SPB   HIGH;
      L     #VAL_0;
      SPA   SAVE;
HIGH: L     #VAL_1;
SAVE: T     #VAL;
      CLR   ;

END_FUNCTION

FUNCTION "m7b_MUXx3xTIME" : TIME
TITLE =3x TIME Multiplexer
//AUTOR: Stefan Maag, Dipl.-Ing. (FH) Elektrotechnik
//DATUM: 10/2008
//INTERNET: www.maagic7.de
//
//AENDERUNGSVERMERKE:
//--------------------------------------------------------------------------------
//DATUM        NAME        AENDERUNG
//--------------------------------------------------------------------------------
//09.10.2008   S.Maag      enstanden aus MUXx3xDINT
//
//24.04.2009   S.Maag      EN0 := Signal Wert selektiert
//                               (S1 | S2 | S3)  AND ENABLE
//
//29.01.2013   S.Maag      Anzeige aktiver Kanal (DSP_CHANNEL)
//--------------------------------------------------------------------------------
//
//HINWEISE:
AUTHOR : 'S.Maag'
FAMILY : Maagic7
VERSION : 0.1


VAR_INPUT
  S1 : BOOL ;
  S2 : BOOL ;
  S3 : BOOL ;
  ENABLE : BOOL ;
  TIME1 : TIME ;
  TIME2 : TIME ;
  TIME3 : TIME ;
END_VAR
VAR_OUTPUT
  DSP_CHANNEL : INT ;	//Displays the activated channel
END_VAR
BEGIN
NETWORK
TITLE =

      UN    #ENABLE; // keine Freigabe, dann 0 ausgeben
      SPB   STOP;

      U     #S1;
      SPB   S1;
      U     #S2;
      SPB   S2;
      U     #S3;
      SPB   S3;

      SPA   STOP;

S1:   L     1; // Wert für Kanalanzeige
      L     #TIME1;
      SPA   SAVE;

S2:   L     2;
      L     #TIME2;
      SPA   SAVE;

S3:   L     3;
      L     #TIME3;
      SPA   SAVE;

STOP: CLR   ; // EN0-Ausgang =0, da Stopp
      L     0; // Wert für Kanalanzeige
      L     T#0MS; // Wert für Multiplexer

SAVE: SAVE  ;
      T     #RET_VAL; // Mulitplexer Ausgang
      TAK   ; // Wert aktiver Kanal
      T     #DSP_CHANNEL; // Anzeige aktiver Kanal

END_FUNCTION

FUNCTION "m7b_MUXx4xTIME" : TIME
TITLE =4x TIME Multiplexer
//AUTOR: Stefan Maag, Dipl.-Ing. (FH) Elektrotechnik
//DATUM: 10/2008
//INTERNET: www.maagic7.de
//
//AENDERUNGSVERMERKE:
//--------------------------------------------------------------------------------
//DATUM        NAME        AENDERUNG
//--------------------------------------------------------------------------------
//09.10.2008   S.Maag      enstanden aus MUXx4xDINT
//
//24.04.2009   S.Maag      EN0 := Signal Wert selektiert
//                               (S1 | S2 | S3)  AND ENABLE
//
//29.01.2013   S.Maag      Anzeige aktiver Kanal (DSP_CHANNEL)
//--------------------------------------------------------------------------------
//
//HINWEISE:
AUTHOR : 'S.Maag'
FAMILY : Maagic7
VERSION : 0.1


VAR_INPUT
  S1 : BOOL ;
  S2 : BOOL ;
  S3 : BOOL ;
  S4 : BOOL ;
  ENABLE : BOOL ;
  TIME1 : TIME ;
  TIME2 : TIME ;
  TIME3 : TIME ;
  TIME4 : TIME ;
END_VAR
VAR_OUTPUT
  DSP_CHANNEL : INT ;	//Displays the activated channel
END_VAR
BEGIN
NETWORK
TITLE =

      UN    #ENABLE; // keine Freigabe, dann 0 ausgeben
      SPB   STOP;

      U     #S1;
      SPB   S1;
      U     #S2;
      SPB   S2;
      U     #S3;
      SPB   S3;
      U     #S4;
      SPB   S4;

      SPA   STOP;

S1:   L     1; // Wert für Kanalanzeige
      L     #TIME1;
      SPA   SAVE;

S2:   L     2;
      L     #TIME2;
      SPA   SAVE;

S3:   L     3;
      L     #TIME3;
      SPA   SAVE;

S4:   L     4;
      L     #TIME4;
      SPA   SAVE;

STOP: CLR   ; // EN0-Ausgang =0, da Stopp
      L     0; // Wert für Kanalanzeige
      L     T#0MS; // Wert für Multiplexer

SAVE: SAVE  ;
      T     #RET_VAL; // Mulitplexer Ausgang
      TAK   ; // Wert aktiver Kanal
      T     #DSP_CHANNEL; // Anzeige aktiver Kanal

END_FUNCTION

FUNCTION "m7b_TOL_TIME" : VOID
TITLE =Wert mit Toleranzbereich ok
//Prüft ob der IST-Wert im Toleranzbereich des Sollwerts ist
//
//AUTOR: Stefan Maag, Dipl.-Ing. (FH) Elektrotechnik
//DATUM: 10/2008
//INTERNET: www.maagic7.de
//
//AENDERUNGSVERMERKE:
//--------------------------------------------------------------------------------
//DATUM        NAME            AENDERUNG
//--------------------------------------------------------------------------------
//09.10.2008  S.Maag      enstanden aus m7TOLERANZ_DINT
//--------------------------------------------------------------------------------
//
//HINWEISE:
AUTHOR : 'S.Maag'
FAMILY : Maagic7
VERSION : 0.1


VAR_INPUT
  IST : TIME ;	//Istwert
  SOLL : TIME ;	//Sollwert
  TOL : TIME ;	//Toleranzbereich
END_VAR
VAR_OUTPUT
  OK : BOOL ;	//Wert im Toleranzbereich
END_VAR
BEGIN
NETWORK
TITLE =

      L     #SOLL; // Sollwert
      L     #IST; // Istwert
      -D    ; // Differenz
      SPP   plus; // Vorzeichen immer
      NEGD  ; // auf positiv
plus: L     #TOL; // Soll, Ist Differenz mit TOL vergleichen
      <=D   ; // ist die ABS(SOLL-IST)<= Toleranz, dann ok!
      =     #OK;
      SAVE  ;
      CLR   ;
END_FUNCTION

FUNCTION "m7b_MIN_MAX_OK_TIME" : VOID
TITLE =Wert zwischen Min und Max? MIN <= VALUE <= MAX
//Prüft ob der IST-Wert zwischen MIN & MAX liegt
//AUTOR: Stefan Maag, Dipl.-Ing. (FH) Elektrotechnik
//DATUM: 10/2008
//INTERNET: www.maagic7.de
//
//AENDERUNGSVERMERKE:
//--------------------------------------------------------------------------------
//DATUM        NAME            AENDERUNG
//--------------------------------------------------------------------------------
//09.10.2008  S.Maag      enstanden aus m7MIN_MAX_OK_DINT
//--------------------------------------------------------------------------------
//
//HINWEISE:
AUTHOR : 'S.Maag'
FAMILY : Maagic7
VERSION : 0.1


VAR_INPUT
  VALUE : TIME ;	//Zu prüfender Wert
  MIN : TIME ;	//Zulässiger Minimalwert
  MAX : TIME ;	//Zulässiger Maximalwert
END_VAR
VAR_OUTPUT
  OK : BOOL ;	//Wert im Toleranzbereich
END_VAR
BEGIN
NETWORK
TITLE =

      L     #MIN; // minmal zulässiger Wert
      L     #VALUE;
      >D    ; // falls MIN > VALUE
      SPB   NOK; // dann nicht ok
      L     #MAX;
      >D    ; // falls VALUE > MAX
      SPB   NOK; // dann nicht ok
      =     #OK; // sonst ok
      SAVE  ;
      BEA   ;
NOK:  CLR   ; // Wert nicht ok
      =     #OK;
      SAVE  ;


END_FUNCTION

FUNCTION "m7b_Scale_TIME" : TIME
TITLE =Bereich Skalieren TIME
//Skaliert eienen Wert von einem Eingagswertebereich auf einen
//Ausgangswertebereich:
//
//FC-ENO: Übersteuerungsanzeige
//
//ACHTUNG: die Eingangswerte werden nicht auf Gültigkeit geprüft
//         und der Ausgangswert wird nicht begrenzt. Bei Übersteuerung wird
//         der FC-ENO-Ausgang "1"
//
//z.B. Eingangswertebereich 100 -  300
//     Ausgangswertebereich   0 - 1000
//
//                           (MaxOutput - MinOutput)
//Xout = (Value - MinInput) --------------------------  + MinOutput
//                            (MaxInput - MinInput)
//
//
//AUTOR: Stefan Maag, Dipl.-Ing. (FH) Elektrotechnik
//DATUM: 3/2003
//INTERNET: www.maagic7.de
//
//AENDERUNGSVERMERKE:
//--------------------------------------------------------------------------------
//DATUM        NAME            AENDERUNG
//--------------------------------------------------------------------------------
//
//--------------------------------------------------------------------------------
//
//HINWEISE:
AUTHOR : 'S.Maag'
FAMILY : Maagic7
VERSION : 0.1


VAR_INPUT
  tMinInput : TIME ;
  tMaxInput : TIME ;
  tValue : TIME ;
  tMinOutput : TIME ;
  tMaxOutput : TIME ;
END_VAR
VAR_TEMP
  rTemp : REAL ;
END_VAR
BEGIN
NETWORK
TITLE =Eingagswertebereich berechnen
//(MaxInput - MinInput)
      L     #tMaxInput;
      L     #tMinInput;
      -D    ; // Differenz
      DTR   ; // zu        REAL
      T     #rTemp;

NETWORK
TITLE =Faktor aus Ausgangs- und Eingangs-Wertebereich
// (MaxOutput - MinOutput)
//-------------------------
//  (MaxInput - MinInput)
      L     #tMaxOutput;
      L     #tMinOutput;
      -D    ; // Differenz
      DTR   ; // zu        REAL
      L     #rTemp;
      /R    ; // Gleitpunktdivision
      T     #rTemp;

NETWORK
TITLE =skalierter Ausgangswert
//                     (MaxOutput - MinOutput)
// (Value - MinInput) -------------------------- + MinOutput
//                      (MaxInput - MinInput)
      L     #tValue; // Eingangswert
      L     #tMinInput; // UnterGrenze Eingangswert
      -D    ; // Differenz
      DTR   ; // zu        REAL
      L     #rTemp;
      *R    ; // Gleitpunktmultiplikation
      RND   ; // zu Festpunkt 32Bit
      L     #tMinOutput;
      +D    ;
      T     #RET_VAL; // Rückgabewert
NETWORK
TITLE =FC-ENO-Ausgangs als Übersteuerungsanzeige

      L     #tMaxOutput; // MaxOutput
      >D    ; // Wert > MaxOutput
      SPB   SAVE; // Max-Wert überschritten
      TAK   ; // Ausgangswert in Akku 1 zurueck
      L     #tMinOutput;
      <D    ;
      SPB   SAVE; // MinWert unterschritten
      CLR   ;
SAVE: SAVE  ;
      CLR   ;
END_FUNCTION

FUNCTION "m7b_MinDiffABS_TIME" : VOID
TITLE =MinDiffABS_TIME: Minimale Absolutdifferenz 2er IEC-Zeiten ok!
//Überprüft, ob die absolute Differenz (absolut) zweier IEC-Zeiten dem
//angebegenen Mindestwert entspricht. Wenn ja, dann wird ENO=True
//
//BENÖTIGTE SFCs: keine
//
//AUTOR: Stefan Maag, Dipl.-Ing. (FH) Elektrotechnik
//DATUM: 3/2008
//INTERNET: www.maagic7.de
//
//AENDERUNGSVERMERKE:
//--------------------------------------------------------------------------------
//DATUM        NAME        AENDERUNG
//--------------------------------------------------------------------------------
//
//--------------------------------------------------------------------------------
//
//HINWEISE:
AUTHOR : 'S.Maag'
FAMILY : Maagic7
VERSION : 0.1


VAR_INPUT
  Time1 : TIME ;
  Time2 : TIME ;
  MinTimeDiff : TIME ;
END_VAR
VAR_TEMP
  aktSysTime : TIME ;	//aktuelle Systemzeit
END_VAR
BEGIN
NETWORK
TITLE =prüfen ob Zeit abgelaufen ist

      L     #Time1;
      L     #Time2;
      -D    ;
      SPP   pos;
      NEGD  ;
pos:  L     #MinTimeDiff;
      >=D   ;
      SAVE  ;

END_FUNCTION

FUNCTION "m7b_SchleppZeiger_TIME" : VOID
TITLE =SchleppZeiger_TIME: Schleppzeiger für TIME (drag indicator)
//Schleppzeiger für IEC-TIME-Werte
//Der FC-ENO-Ausgang wird dann "1", wenn der Schleppzeiger einen neuen Wert
//erhält, ansonsten ist der FC-ENO-Ausgang "0"
//
//AUTOR: Stefan Maag, Dipl.-Ing. (FH) Elektrotechnik
//DATUM: 9/2004
//INTERNET: www.maagic7.de
//
//AENDERUNGSVERMERKE:
//--------------------------------------------------------------------------------
//DATUM        NAME            AENDERUNG
//--------------------------------------------------------------------------------
//
//--------------------------------------------------------------------------------
//
//HINWEISE:
AUTHOR : 'S.Maag'
FAMILY : Maagic7
VERSION : 0.1


VAR_INPUT
  tValue : TIME ;	//aktueller Wert
  cfgMinMax : BOOL ;	//Konfig.: 0=Minimum Schleppzeiger 1=Maximum Schleppzeiger
  Init : BOOL ;	//Initialisierung, Schleppzeiger wird auf aktuellen Wert gesetzt
END_VAR
VAR_IN_OUT
  SchleppZeiger : TIME ;	//Schleppzeiger-Wert
END_VAR
BEGIN
NETWORK
TITLE =

      U     #Init;
      SPB   INIT;

      U     #cfgMinMax; // Maximum Schleppzeiger
      SPB   MAX;

      L     #SchleppZeiger; // Minimum Schleppzeiger
      L     #tValue;
      <D    ;
      SPB   END;
      SPA   SAVE;

INIT: L     #tValue; // Schleppzeicher initialisieren
      SPA   SAVE;

MAX:  L     #SchleppZeiger;
      L     #tValue;
      >D    ;
      SPB   END;

SAVE: T     #SchleppZeiger;
      SET   ;
      SAVE  ;
      CLR   ;
      BEA   ;

END:  CLR   ;
      SAVE  ;

END_FUNCTION

FUNCTION "m7b_ChangeEvent_TOD" : VOID
TITLE =Ereignis Time_Of_Day Wert hat sich geändert
//Der FC-ENO-Ausgang wird für einen Zyklus "1", wenn der sich der Eingangswert
//geändert hat, ansonsten ist der FC-ENO-Ausgang "0"
//
//AUTOR: Stefan Maag, Dipl.-Ing. (FH) Elektrotechnik
//DATUM: 10/2008
//INTERNET: www.maagic7.de
//
//AENDERUNGSVERMERKE:
//--------------------------------------------------------------------------------
//DATUM        NAME            AENDERUNG
//--------------------------------------------------------------------------------
//
//--------------------------------------------------------------------------------
//
//HINWEISE:
AUTHOR : 'S.Maag'
FAMILY : Maagic7
VERSION : 0.1


VAR_INPUT
  inTOD : TIME_OF_DAY ;
END_VAR
VAR_IN_OUT
  memTOD : TIME_OF_DAY ;
END_VAR
BEGIN
NETWORK
TITLE =

      L     #inTOD; // Eingangwert
      L     #memTOD; // letzter Wert
      <>D   ; // ungleich!
      SAVE  ; // als ENO ausgeben
      SPB   do; // und neuen
      BEA   ;
do:   L     #inTOD; // Wert speichern
      T     #memTOD;

END_FUNCTION

FUNCTION "m7b_MinMaxLimit_TOD" : VOID
TITLE =Min/Max limit Time_Of_Day; Begrenzungsanzeige im BIE-Bit/FC-ENO
//Min- Max- Begrenzung für TIME mit Begrenzungsanzeige
//
//BIE bzw. FC-ENO : 0 = Wert war ok       : Begrenzung nicht aktiv
//                  1 = Wert war nicht ok.: Begrenzung aktiv
//
//AUTOR: Stefan Maag, Dipl.-Ing. (FH) Elektrotechnik
//DATUM: 10/2008
//INTERNET: www.maagic7.de
//
//VERWENDUNG:
//Begrenzung eines Wertes auf den Min- Max- Bereich bei gleichzeitiger
//Weiterverarbeitung des Begrenzungssignals am FC-ENO-Ausgang z.B. zur Warn- bzw.
//Störungsanzeige oder zur direkten Weiterverschaltung.
//
//AENDERUNGSVERMERKE:
//--------------------------------------------------------------------------------
//DATUM        NAME            AENDERUNG
//--------------------------------------------------------------------------------
//
//--------------------------------------------------------------------------------
//
//HINWEISE:
AUTHOR : 'S.Maag'
FAMILY : Maagic7
VERSION : 0.1


VAR_INPUT
  min : TIME_OF_DAY ;	//minimal Wert
  max : TIME_OF_DAY ;	//maximal Wert
END_VAR
VAR_IN_OUT
  VALUE : TIME_OF_DAY ;	//Sollwert
END_VAR
BEGIN
NETWORK
TITLE =MIN <= VALUE <= MAX

      L     #VALUE; // Sollwert
      L     #min; // minimal Wert
      <D    ;
      SPB   LIM; // Limitierung wenn VALUE < MIN
      TAK   ; // VALUE wieder in Akku 1
      L     #max; // Maximalwert
      >D    ;
      SPB   LIM; // Limitierung wenn VALUE > MAX

      CLR   ; // VKE löschen, da keine Begrenzung erfolgte
      SAVE  ; // BIE-Bit = 0, da Wert im Bereich war; ="Keine Begrenzung"
      BEA   ;

LIM:  T     #VALUE; // max.Wert als Sollwert ausgeben
      SET   ;
      SAVE  ; // VKE->BIE (=1=): Anzeige FC-ENO Ausgang (=Begrenzung)
      CLR   ;

END_FUNCTION

FUNCTION "m7b_BitToTOD" : VOID
TITLE =Bit To Time_Of_Day
//Je nach dem Wert des Eingangsbits wird der Wert
//VAL_0 oder VAL_1 als Ausgangswert VAL ausgegeben.
//Der Wert der Eingangsbits wird auf den FC-ENO-Ausgang durchgeschleift
//
//AUTOR: Stefan Maag, Dipl.-Ing. (FH) Elektrotechnik
//DATUM: 10/2008
//
//AENDERUNGSVERMERKE:
//--------------------------------------------------------------------------------
//DATUM        NAME            AENDERUNG
//--------------------------------------------------------------------------------
//
//--------------------------------------------------------------------------------
//
//HINWEISE:
AUTHOR : 'S.Maag'
FAMILY : Maagic7
VERSION : 0.1


VAR_INPUT
  BIT : BOOL ;
  VAL_0 : TIME_OF_DAY ;
  VAL_1 : TIME_OF_DAY ;
END_VAR
VAR_OUTPUT
  VAL : TIME ;
END_VAR
BEGIN
NETWORK
TITLE =

      U     #BIT;
      SAVE  ; // Wert von Bit auf FC-EN0
      SPB   HIGH;
      L     #VAL_0;
      SPA   SAVE;
HIGH: L     #VAL_1;
SAVE: T     #VAL;
      CLR   ;

END_FUNCTION

FUNCTION "m7b_MUXx3xTOD" : TIME_OF_DAY
TITLE =3x Time_Of_Day Multiplexer
//AUTOR: Stefan Maag, Dipl.-Ing. (FH) Elektrotechnik
//DATUM: 10/2008
//INTERNET: www.maagic7.de
//
//AENDERUNGSVERMERKE:
//--------------------------------------------------------------------------------
//DATUM        NAME        AENDERUNG
//--------------------------------------------------------------------------------
//09.10.2008   S.Maag      enstanden aus MUXx3xDINT
//
//24.04.2009   S.Maag      EN0 := Signal Wert selektiert
//                               (S1 | S2 | S3)  AND ENABLE
//
//29.01.2013   S.Maag      Anzeige aktiver Kanal (DSP_CHANNEL)
//--------------------------------------------------------------------------------
//
//HINWEISE:
AUTHOR : 'S.Maag'
FAMILY : Maagic7
VERSION : 0.1


VAR_INPUT
  S1 : BOOL ;
  S2 : BOOL ;
  S3 : BOOL ;
  ENABLE : BOOL ;
  TIME1 : TIME_OF_DAY ;
  TIME2 : TIME_OF_DAY ;
  TIME3 : TIME_OF_DAY ;
END_VAR
VAR_OUTPUT
  DSP_CHANNEL : INT ;	//Displays the activated channel
END_VAR
BEGIN
NETWORK
TITLE =

      UN    #ENABLE; // keine Freigabe, dann 0 ausgeben
      SPB   STOP;

      U     #S1;
      SPB   S1;
      U     #S2;
      SPB   S2;
      U     #S3;
      SPB   S3;

      SPA   STOP;

S1:   L     1; // Wert für Kanalanzeige
      L     #TIME1;
      SPA   SAVE;

S2:   L     2;
      L     #TIME2;
      SPA   SAVE;

S3:   L     3;
      L     #TIME3;
      SPA   SAVE;


STOP: CLR   ; // EN0-Ausgang =0, da Stopp
      L     0; // Wert für Kanalanzeige
      L     L#0; // Wert für Multiplexer

SAVE: SAVE  ;
      T     #RET_VAL; // Mulitplexer Ausgang
      TAK   ; // Wert aktiver Kanal
      T     #DSP_CHANNEL; // Anzeige aktiver Kanal

END_FUNCTION

FUNCTION "m7b_MUXx4xTOD" : TIME_OF_DAY
TITLE =4x Time_Of_Day Multiplexer
//AUTOR: Stefan Maag, Dipl.-Ing. (FH) Elektrotechnik
//DATUM: 10/2008
//INTERNET: www.maagic7.de
//
//AENDERUNGSVERMERKE:
//--------------------------------------------------------------------------------
//DATUM        NAME        AENDERUNG
//--------------------------------------------------------------------------------
//09.10.2008   S.Maag      enstanden aus MUXx4xDINT
//
//24.04.2009   S.Maag      EN0 := Signal Wert selektiert
//                               (S1 | S2 | S3)  AND ENABLE
//
//29.01.2013   S.Maag      Anzeige aktiver Kanal (DSP_CHANNEL)
//--------------------------------------------------------------------------------
//
//HINWEISE:
AUTHOR : 'S.Maag'
FAMILY : Maagic7
VERSION : 0.1


VAR_INPUT
  S1 : BOOL ;
  S2 : BOOL ;
  S3 : BOOL ;
  S4 : BOOL ;
  ENABLE : BOOL ;
  TIME1 : TIME_OF_DAY ;
  TIME2 : TIME_OF_DAY ;
  TIME3 : TIME_OF_DAY ;
  TIME4 : TIME_OF_DAY ;
END_VAR
VAR_OUTPUT
  DSP_CHANNEL : INT ;	//Displays the activated channel
END_VAR
BEGIN
NETWORK
TITLE =

      UN    #ENABLE; // keine Freigabe, dann 0 ausgeben
      SPB   STOP;

      U     #S1;
      SPB   S1;
      U     #S2;
      SPB   S2;
      U     #S3;
      SPB   S3;
      U     #S4;
      SPB   S4;

      SPA   STOP;

S1:   L     1; // Wert für Kanalanzeige
      L     #TIME1;
      SPA   SAVE;

S2:   L     2;
      L     #TIME2;
      SPA   SAVE;

S3:   L     3;
      L     #TIME3;
      SPA   SAVE;

S4:   L     4;
      L     #TIME4;
      SPA   SAVE;

STOP: CLR   ; // EN0-Ausgang =0, da Stopp
      L     0; // Wert für Kanalanzeige
      L     L#0; // Wert für Multiplexer

SAVE: SAVE  ;
      T     #RET_VAL; // Mulitplexer Ausgang
      TAK   ; // Wert aktiver Kanal
      T     #DSP_CHANNEL; // Anzeige aktiver Kanal

END_FUNCTION

FUNCTION "m7b_TOL_TOD" : VOID
TITLE =Wert mit Toleranzbereich ok [Time_Of_Day]
//Prüft ob der IST-Wert im Toleranzbereich des Sollwerts ist
//ACHTUNG: Die Toleranz kann nicht als Tageszeit angegeben werden, sie ist als
//         TIME anzugeben
//
//AUTOR: Stefan Maag, Dipl.-Ing. (FH) Elektrotechnik
//DATUM: 10/2008
//INTERNET: www.maagic7.de
//
//AENDERUNGSVERMERKE:
//--------------------------------------------------------------------------------
//DATUM        NAME            AENDERUNG
//--------------------------------------------------------------------------------
//09.10.2008  S.Maag      enstanden aus m7TOLERANZ_DINT
//--------------------------------------------------------------------------------
//
//HINWEISE:
AUTHOR : 'S.Maag'
FAMILY : Maagic7
VERSION : 0.1


VAR_INPUT
  IST : TIME_OF_DAY ;	//Istwert
  SOLL : TIME_OF_DAY ;	//Sollwert
  TOL : TIME ;	//Toleranzbereich
END_VAR
VAR_OUTPUT
  OK : BOOL ;	//Wert im Toleranzbereich
END_VAR
BEGIN
NETWORK
TITLE =

      L     #SOLL; // Sollwert
      L     #IST; // Istwert
      -D    ; // Differenz
      SPP   plus; // Vorzeichen immer
      NEGD  ; // auf positiv
plus: L     #TOL; // Soll, Ist Differenz mit TOL vergleichen
      <=D   ; // ist die ABS(SOLL-IST)<= Toleranz, dann ok!
      =     #OK;
      SAVE  ;
      CLR   ;
END_FUNCTION

FUNCTION "m7b_MIN_MAX_OK_TOD" : VOID
TITLE =Wert zwischen Min und Max? MIN <= VALUE <= MAX
//Prüft ob der IST-Wert zwischen MIN & MAX liegt
//AUTOR: Stefan Maag, Dipl.-Ing. (FH) Elektrotechnik
//DATUM: 10/2008
//INTERNET: www.maagic7.de
//
//AENDERUNGSVERMERKE:
//--------------------------------------------------------------------------------
//DATUM        NAME            AENDERUNG
//--------------------------------------------------------------------------------
//09.10.2008  S.Maag      enstanden aus m7MIN_MAX_OK_DINT
//--------------------------------------------------------------------------------
//
//HINWEISE:
AUTHOR : 'S.Maag'
FAMILY : Maagic7
VERSION : 0.1


